	2:  (*Produktions Meldung*)
		Visu.MeldungProduktion.Color_R := 255;
		Visu.MeldungProduktion.Color_G := 255;
		Visu.MeldungProduktion.Color_B := 0;
		IF visu.s_akt_sprache = 'de' THEN
			Visu.MeldungProduktion.Name:='Y-Achse WT Übergabepos größer als Endlage';
		ELSIF visu.s_akt_sprache = 'en' THEN
			Visu.MeldungProduktion.Name:='Y-Achse WT Übergabepos größer als Endlage';
		ELSIF visu.s_akt_sprache = 'cz' THEN
			Visu.MeldungProduktion.Name:='Y-Achse WT Übergabepos größer als Endlage';
		END_IF
		Visu.MeldungProduktion.ShowMessage := TRUE;
		Visu.MeldungProduktion.Button1.sichtbar:= FALSE;	(*OK*)
		Visu.MeldungProduktion.Button1.Text:='Ok';
		i16_state_msg := 3;

	3:  (*Warte auf OK*)
		IF NOT b_EndlageErreicht THEN
			ST_Message_Produktion.b_PM_Quitt:=TRUE;
			i16_state_msg:=0;
		END_IF
END_CASE

(* =======================================Toplevel========================================== *)
(* Starte Inbetriebnahme-Sequenz *)
IF st_ctrl_in.b_gehe_step_ibn THEN
	fb_state_entry.i16_next_step := INBETRIEBNAHME;
END_IF

(* =====Achse wird disabled===== *)
IF (NOT e_steuerung_ein OR NOT e_ba_mit_bedingungen) AND y_achse.Status.Operational THEN
	st_drive_cmd.enu_cmd := POWER_DISABLE;
END_IF

IF fb_state_entry.i16_next_step > INIT AND fb_state_entry.i16_next_step < FEHLER THEN
	(* =====Fehler vom Achskontroller===== *)
	IF st_drive_cmd.b_job_fehler THEN
		fb_state_entry.i16_next_step := FEHLER;
	END_IF

	IF fb_state_entry.i16_next_step > 35 THEN
		(* Devicefehler *)
		IF y_achse.Status.Error THEN
			st_sm.b_achsfehler := TRUE;
			fb_state_entry.i16_next_step := FEHLER;
		ELSIF y_achse.Status.DriveDeviceError THEN
			st_sm.b_devicefehler := TRUE;
			fb_state_entry.i16_next_step := FEHLER;
		END_IF
	END_IF

	IF fb_state_entry.i16_next_step < STOP THEN
		(* =====Achse wird gestoppt===== *)
		IF st_ctrl_in.b_stop THEN
			fb_state_entry.i16_next_step := STOP;
		ELSIF fb_state_entry.i16_next_step < HALT THEN
			(* =====Achse wird angehalten===== *)
			IF st_ctrl_in.b_halt THEN
				fb_state_entry.i16_next_step := HALT;
			END_IF
		END_IF
	END_IF
END_IF

(* ======================================Schrittkette======================================== *)
fb_state_entry(
	i16_next_step:= ,
	i16_pos:= 1,
	E=> ,
	X=> , 
	i16_step=> ,
	i16_last_step=> );

CASE fb_state_entry.i16_step OF
(*=======================================================*)
	INIT_OBJ:
		IF st_config_achse.b_config_fertig THEN
			fb_state_entry.i16_next_step := 1;
		END_IF

(*=======================================================*)
	1:	(* Warte bis NetID´s der Slaves ausgelesen sind *)
		IF fb_state_entry.E THEN
			;
		END_IF

		(*-----------------------Weiterschaltbedingungen----------------------------*)
		IF ST_EthercatDiag.st_ctrl_out.b_fertig THEN
			fb_state_entry.i16_next_step := 2;
		END_IF

(*=======================================================*)
	2:	(* Spezifische NC-Achsparameter auslesen *)
		IF fb_state_entry.E THEN
			fb_axis.i16_nc_parameter_nummer := MaxVelocitySystem;
			st_drive_cmd.enu_cmd := READ_NC_PARAMETER;
		END_IF

		(*-----------------------Weiterschaltbedingungen----------------------------*)
		IF st_drive_cmd.enu_cmd = NO_COMMAND THEN
			lr_Velo_in:=st_geschwindigkeiten.lr_maximalgeschwindigkeit;
			st_geschwindigkeiten.lr_auto_max := st_geschwindigkeiten.lr_maximalgeschwindigkeit := fb_axis.r_wert_nc_read_parameter;
			st_geschwindigkeiten.lr_auto_min := 25.0;
			st_geschwindigkeiten.lr_jog := 50;
			fb_state_entry.i16_next_step := 3;
		END_IF

(*=======================================================*)
	3:	(* Spezifische NC-Achsparameter auslesen *)
		IF fb_state_entry.E THEN
			fb_axis.i16_nc_parameter_nummer := MaxAccelerationSystem;
			st_drive_cmd.enu_cmd := READ_NC_PARAMETER;
		END_IF

		(*-----------------------Weiterschaltbedingungen----------------------------*)
		IF st_drive_cmd.enu_cmd = NO_COMMAND THEN
			st_geschwindigkeiten.lr_beschleunigung := fb_axis.r_wert_nc_read_parameter;
			fb_state_entry.i16_next_step := 4;
		END_IF

(*=======================================================*)
	4:	(* Spezifische NC-Achsparameter auslesen *)
		IF fb_state_entry.E THEN
			fb_axis.i16_nc_parameter_nummer := MaxDecelerationSystem;
			st_drive_cmd.enu_cmd := READ_NC_PARAMETER;
		END_IF

		(*-----------------------Weiterschaltbedingungen----------------------------*)
		IF st_drive_cmd.enu_cmd = NO_COMMAND THEN
			st_geschwindigkeiten.lr_verzoegerung := fb_axis.r_wert_nc_read_parameter;
			lr_decceleration_normal := st_geschwindigkeiten.lr_verzoegerung;
			lr_decceleration_nothalt := 200000.0;
			fb_state_entry.i16_next_step := 5;
		END_IF

(*=======================================================*)
	5:	(* Spezifische NC-Achsparameter auslesen *)
		IF fb_state_entry.E THEN
			fb_axis.i16_nc_parameter_nummer := MaxJerk;
			st_drive_cmd.enu_cmd := READ_NC_PARAMETER;
		END_IF

		(*-----------------------Weiterschaltbedingungen----------------------------*)
		IF st_drive_cmd.enu_cmd = NO_COMMAND THEN
			st_geschwindigkeiten.lr_ruck := fb_axis.r_wert_nc_read_parameter;
			fb_state_entry.i16_next_step := 6;
		END_IF

(*=======================================================*)
	6:	(* Konfigurationen der Achse *)
		IF fb_state_entry.E THEN
			fb_axis.st_eccoe_sdo.s_ec_slave_net_id := ST_EthercatDiag.s_ec_slave_net_id[2];
			fb_axis.st_eccoe_sdo.ui16_slave_addr := st_config_achse.ui16_ethercat_adr;
		END_IF

		(*-----------------------Weiterschaltbedingungen----------------------------*)
		fb_state_entry.i16_next_step := 7;

(*=======================================================*)
	7:	(* Spezifische NC-Achsparameter auslesen *)
		IF fb_state_entry.E THEN
			fb_axis.i16_nc_parameter_nummer := AxisMinSoftPosLimit;
			st_drive_cmd.enu_cmd := READ_NC_PARAMETER;
		END_IF

		(*-----------------------Weiterschaltbedingungen----------------------------*)
		IF st_drive_cmd.enu_cmd = NO_COMMAND THEN
			lr_MinSoftPosLimit := fb_axis.r_wert_nc_read_parameter;
			fb_state_entry.i16_next_step := 8;
		END_IF


(*=======================================================*)
	8:	(* Spezifische NC-Achsparameter auslesen *)
		IF fb_state_entry.E THEN
			fb_axis.i16_nc_parameter_nummer := AxisMaxSoftPosLimit;
			st_drive_cmd.enu_cmd := READ_NC_PARAMETER;
		END_IF

		(*-----------------------Weiterschaltbedingungen----------------------------*)
		IF st_drive_cmd.enu_cmd = NO_COMMAND THEN
			lr_MaxSoftPosLimit := fb_axis.r_wert_nc_read_parameter;
			fb_state_entry.i16_next_step := FEHLER; (*in Fehler gehen damit die Achsen resetet werden. Sonst steigen die Achsen bei einem TC Restart aus*)
		END_IF

(*=======================================================*)
	INIT:
		IF fb_state_entry.E THEN
			fb_ton_wz.IN := FALSE;
			fb_ton_uez.IN	:= FALSE;
			fb_ton_quitt.IN := FALSE;
			(* Reset Stoermeldungen *)
			st_sm.b_achse_nicht_auf_startpos := FALSE;
			st_sm.b_achsfehler := FALSE;
			st_sm.b_devicefehler := FALSE;
			st_sm.b_keine_verfahrfreigabe := FALSE;
			st_sm.b_ende_skalierungs_nocke := FALSE;
			st_sm.b_ende_camming_nocke := FALSE;
			st_sm.b_skalierung_noch_aktiv := FALSE;
			b_start_in:=FALSE;
			st_ctrl_out.b_busy:=FALSE;
			st_ctrl_out.b_fehler := FALSE;
			st_ctrl_out.b_fertig := FALSE;

			st_ctrl_out.b_bereit := FALSE;
			st_ctrl_out.b_prebereit := FALSE;
			sm_kein_nocken_definiert := FALSE;

			fb_axis.lr_soll_geschwindigkeit := gst_datensatz.st_wkz.r_auto_y;

			st_geschwindigkeiten.lr_verzoegerung := lr_decceleration_normal;
		END_IF

		(*-----------------------Weiterschaltbedingungen----------------------------*)
		IF st_ctrl_in.b_preinit THEN
			fb_state_entry.i16_next_step := 15;
		END_IF

(*=======================================================*)
	15:	(* Reglerfreigabe wegnehmen *)
		IF fb_state_entry.E THEN
			st_drive_cmd.enu_cmd := POWER_DISABLE;
		END_IF

		(*-----------------------Weiterschaltbedingungen----------------------------*)
		IF st_drive_cmd.enu_cmd = NO_COMMAND THEN
			fb_state_entry.i16_next_step := 20;
		END_IF

(*=======================================================*)
	20:	(* Überprüfe Nullpunktverschiebung des Absolutwertgebers auf Korrektheit *)
		IF fb_state_entry.E THEN
			fb_axis.i16_nc_parameter_nummer := AxisEncoderOffset;	(* vom Datentyp MC_AxisParameter *)
			st_drive_cmd.enu_cmd := READ_NC_PARAMETER;
		END_IF

		(*-----------------------Weiterschaltbedingungen----------------------------*)
		IF st_drive_cmd.enu_cmd = NO_COMMAND THEN
			IF fb_axis.r_wert_nc_read_parameter = gst_datensatz.st_md.st_md_y_achse.lr_nullpunktverschiebung THEN
				fb_state_entry.i16_next_step := 35;	(* Reglerfreigabe setzen *)
			ELSE
				fb_state_entry.i16_next_step := 25;	(* Nullpunktverschiebung schreiben *)
			END_IF
		END_IF

(*=======================================================*)
	25:	(* Nullpunktverschiebung hat sich geändert, deshalb erst Null reinschreiben, um keinen Additionsfehler zu machen, *)
		(* weil der Wert der Verschiebung beim Neustart komplett auf die Achse geschrieben wird *)
		IF fb_state_entry.E THEN
			fb_axis.i16_nc_parameter_nummer := AxisEncoderOffset;
			fb_axis.r_wert_nc_write_parameter := 0.0;
			st_drive_cmd.enu_cmd := WRITE_NC_PARAMETER;
		END_IF

		(*-----------------------Weiterschaltbedingungen----------------------------*)
		IF st_drive_cmd.enu_cmd = NO_COMMAND THEN
			fb_state_entry.i16_next_step := 30;
		END_IF

(*=======================================================*)
	30:	(* Aktuelle Nullpunktverschiebung des Absolutwertgebers an die Achse senden *)
		IF fb_state_entry.E THEN
			fb_axis.i16_nc_parameter_nummer := AxisEncoderOffset;
			fb_axis.r_wert_nc_write_parameter := gst_datensatz.st_md.st_md_y_achse.lr_nullpunktverschiebung;
			st_drive_cmd.enu_cmd := WRITE_NC_PARAMETER;
		END_IF

		(*-----------------------Weiterschaltbedingungen----------------------------*)
		IF st_drive_cmd.enu_cmd = NO_COMMAND THEN
			fb_state_entry.i16_next_step := 35;
		END_IF

(*=======================================================*)
	35:	(* Reglerfreigabe setzen , Reset wird bei Bedarf automatisch ausgeführt*)
		IF fb_state_entry.E THEN
			st_drive_cmd.enu_cmd := POWER_ENABLE;
		END_IF

		(*-----------------------Weiterschaltbedingungen----------------------------*)
		IF st_drive_cmd.enu_cmd = NO_COMMAND THEN
			fb_state_entry.i16_next_step := 40;
		END_IF

(*=======================================================*)
	40:	(* Nullpunktverschiebung ist geschrieben *)
		IF fb_state_entry.E THEN
			st_ctrl_out.b_prebereit := TRUE;
		END_IF

		(*-----------------------Weiterschaltbedingungen----------------------------*)
		IF st_ctrl_in.b_init THEN
			fb_state_entry.i16_next_step := 45;
		END_IF

(*=======================================================*)
	45: (* Warte auf Startsignal zum Positionieren *)

		(*-----------------------Weiterschaltbedingungen----------------------------*)
		IF st_ctrl_in.b_start THEN
			fb_state_entry.i16_next_step := 50;
		END_IF

(*=======================================================*)
	50: (* Positioniere Achse auf ausgelesene Slaveposition *)
		IF fb_state_entry.E THEN
			fb_axis.st_position.r_soll := ST_Z_Achse.lr_slave_position;
			st_drive_cmd.enu_cmd := MOVE_ABSOLUTE;
		END_IF

		(*-----------------------Weiterschaltbedingungen----------------------------*)
		IF st_drive_cmd.enu_cmd = NO_COMMAND THEN
			fb_state_entry.i16_next_step := 60;
		END_IF

(*=======================================================*)
	60: (* Warte bis Y-Achse gekoppelt wurde *)
		IF fb_state_entry.E THEN
			st_ctrl_out.b_fertig := TRUE;
		END_IF

		(*-----------------------Weiterschaltbedingungen----------------------------*)
		IF y_achse.NcToPlc.CoupleState = 3 THEN
			st_ctrl_out.b_fertig := FALSE;
			fb_state_entry.i16_next_step := BEREIT;
		END_IF

(*=======================================================*)
	BEREIT:
		IF fb_state_entry.E THEN
			st_ctrl_out.b_bereit := TRUE;
			enu_cmd_in:=NO_COMMAND;
		END_IF

		(*-----------------------Weiterschaltbedingungen----------------------------*)
		IF fb_r_trig_start.Q THEN
			st_ctrl_out.b_fertig_2 := FALSE;
			fb_state_entry.i16_next_step := 110;
		END_IF

		IF 	fb_r_trig_start_in.Q THEN		(*neu! zum Starten einer Positionierung von einem externen Prg.*)
			st_ctrl_out.b_fertig := FALSE;
			fb_state_entry.i16_next_step := 102;
		END_IF

		IF fb_state_entry.X THEN
			st_ctrl_out.b_fertig := FALSE;
			st_ctrl_out.b_busy:=TRUE;
		END_IF

(*=======================================================*)
	102:
		IF 	fb_state_entry.E THEN
			b_start_in:=FALSE;
		END_IF

		(*-----------------------Weiterschaltbedingungen----------------------------*)
		IF 	st_drive_cmd.enu_cmd = NO_COMMAND THEN
			fb_state_entry.i16_next_step := 104;
		END_IF

(*=======================================================*)
	104: (* Positioniere Achse  *)
		IF 	fb_state_entry.E THEN
			fb_axis.st_position.r_soll := lr_Achspos_in ;
			fb_axis.lr_soll_geschwindigkeit:=lr_Velo_in;
			st_drive_cmd.enu_cmd := enu_cmd_in;
		END_IF

		(*-----------------------Weiterschaltbedingungen----------------------------*)
		IF 	st_drive_cmd.enu_cmd = NO_COMMAND THEN
			st_ctrl_out.b_fertig := TRUE;
			fb_state_entry.i16_next_step := BEREIT;
		END_IF

		IF 	fb_state_entry.X THEN
			st_ctrl_out.b_busy:=FALSE;
		END_IF

(*=======================================================*)
	110: (* Fallunterscheidung *)
		CASE gst_datensatz.st_md.i16_typ_zelle OF
			KEINE_ZELLE:
				;

			BESTUECKZELLE_1700:
				(*-----------------------Weiterschaltbedingungen----------------------------*)
				fb_state_entry.i16_next_step := 200;

			RASTERFOLIE:
				(*-----------------------Weiterschaltbedingungen----------------------------*)
				fb_state_entry.i16_next_step := 120;

		END_CASE

(*=======================================================*)
	120: (* Positioniere Achse auf  0-Koordinate  des ISK *)
		IF fb_state_entry.E THEN
			fb_axis.st_position.r_soll := 	gst_datensatz.st_isk.lr_pos_y_0 +
										gst_datensatz.st_wkz.lr_offset_y_pos_0 +
										gst_datensatz.st_wt.lr_offset_y_pos_0 +
										gst_datensatz.st_md.lr_offset_y_pos_0 +
										gst_datensatz.st_bestueckprogramm.lr_y[0];
			st_drive_cmd.enu_cmd := MOVE_ABSOLUTE;
		END_IF

		(*-----------------------Weiterschaltbedingungen----------------------------*)
		IF st_drive_cmd.enu_cmd = NO_COMMAND THEN
			st_ctrl_out.b_fertig := TRUE;
			st_ctrl_out.b_busy:=FALSE;
			fb_state_entry.i16_next_step := 300;
		END_IF

(*=======================================================*)
	200:
		IF fb_state_entry.E THEN
			st_ctrl_out.b_fertig := TRUE;
			st_ctrl_out.b_busy:=FALSE;
		END_IF

		(*-----------------------Weiterschaltbedingungen----------------------------*)
		IF st_ctrl_in.b_start_2 THEN
			st_ctrl_out.b_fertig := FALSE;
			fb_state_entry.i16_next_step := 210;
		END_IF

(*=======================================================*)
	210: (* Positioniere Achse auf gewünschte Position *)
		IF fb_state_entry.E THEN
			fb_axis.st_position.r_soll :=  ST_Z_Achse.lr_slave_position;
			st_drive_cmd.enu_cmd := MOVE_ABSOLUTE;
		END_IF

		(*-----------------------Weiterschaltbedingungen----------------------------*)
		IF st_drive_cmd.enu_cmd = NO_COMMAND THEN
			fb_state_entry.i16_next_step := 220;
		END_IF

(*=======================================================*)
	220: (* Warte bis Y-Achse gekoppelt wurde *)
		IF fb_state_entry.E THEN
			st_ctrl_out.b_fertig_2 := TRUE;
		END_IF

		(*-----------------------Weiterschaltbedingungen----------------------------*)
		IF y_achse.NcToPlc.CoupleState = 3 THEN
			st_ctrl_out.b_fertig_2 := FALSE;
			fb_state_entry.i16_next_step := BEREIT;
		END_IF

(*=======================================================*)
	300:(* Verfahre Y-Achse undwarte auf Start von Z-Achse *)

		(*-----------------------Weiterschaltbedingungen----------------------------*)
		(* Verfahre Y-Achse *)
		IF	gst_datensatz.st_md.i16_typ_zelle = RASTERFOLIE AND
			ST_Rasterfolienmontage.b_start_y_Achse THEN
			fb_state_entry.i16_next_step := 310;
		END_IF

		(* Warte auf Start von Z-Achse *)
		IF st_ctrl_in.b_start_2 THEN
			st_ctrl_out.b_fertig := FALSE;
			fb_state_entry.i16_next_step := 350;
		END_IF

(*=======================================================*)
	310: (* Positioniere Achse  *)
		IF fb_state_entry.E THEN
			fb_axis.st_position.r_soll := 	lr_tmp_Achspos;
			st_drive_cmd.enu_cmd := MOVE_ABSOLUTE;
		END_IF

		(*-----------------------Weiterschaltbedingungen----------------------------*)
		IF st_drive_cmd.enu_cmd = NO_COMMAND THEN
			fb_state_entry.i16_next_step := 300;
			ST_Rasterfolienmontage.b_start_y_Achse:=FALSE;
		END_IF


(*=======================================================*)
	350: (* Positioniere Achse auf gewünschte Position am Ende der Kurvenscheibe *)
		IF fb_state_entry.E THEN
			fb_axis.st_position.r_soll :=  ST_Z_Achse.lr_slave_position;
			st_drive_cmd.enu_cmd := MOVE_ABSOLUTE;
		END_IF

		(*-----------------------Weiterschaltbedingungen----------------------------*)
		IF st_drive_cmd.enu_cmd = NO_COMMAND THEN
			fb_state_entry.i16_next_step := 360;
		END_IF

(*=======================================================*)
	360: (* Warte bis Y-Achse gekoppelt wurde *)
		IF fb_state_entry.E THEN
			st_ctrl_out.b_fertig_2 := TRUE;
		END_IF

		(*-----------------------Weiterschaltbedingungen----------------------------*)
		IF y_achse.NcToPlc.CoupleState = 3 THEN
			st_ctrl_out.b_fertig_2 := FALSE;
			fb_state_entry.i16_next_step := BEREIT;
		END_IF

(*=======================================================*)
	FEHLER:
		IF fb_state_entry.E THEN
			st_ctrl_out.b_fehler := TRUE;
			fb_ton_quitt.IN := FALSE;
			st_ctrl_out.b_busy:=FALSE;
		END_IF

		IF st_ctrl_in.b_stop AND NOT y_achse.Status.HasBeenStopped THEN
			st_drive_cmd.enu_cmd := STOP_AXIS;
		END_IF

		IF st_ctrl_in.b_halt AND y_achse.Status.Moving THEN
			st_drive_cmd.enu_cmd := HALT_AXIS;
			st_geschwindigkeiten.lr_verzoegerung := lr_decceleration_nothalt;
		END_IF

		(*-----------------------Weiterschaltbedingungen----------------------------*)
		IF st_ctrl_in.b_quitt AND NOT fb_state_entry.E THEN
			st_ctrl_out.b_fehler := FALSE;
			st_drive_cmd.enu_cmd := RESET;
			fb_ton_quitt.IN := TRUE;
		END_IF

		IF fb_ton_quitt.Q THEN
			fb_ton_quitt.IN := FALSE;
			fb_state_entry.i16_next_step := INIT;
		END_IF

(*=======================================================*)
	STOP:
		IF fb_state_entry.E THEN
			st_ctrl_out.b_busy:=FALSE;
			IF y_achse.NcToPlc.CoupleState = 0 THEN
				st_drive_cmd.enu_cmd := STOP_AXIS;
			END_IF
		END_IF

		(*-----------------------Weiterschaltbedingungen----------------------------*)
		IF st_drive_cmd.enu_cmd = NO_COMMAND AND y_achse.Status.NotMoving THEN
			fb_state_entry.i16_next_step := STILLSTAND;
		END_IF

(*=======================================================*)
	STILLSTAND:
		IF fb_state_entry.E THEN
			st_drive_cmd.enu_cmd := POWER_DISABLE;
			fb_ton_quitt.IN := FALSE;
		END_IF

		(*-----------------------Weiterschaltbedingungen----------------------------*)
		IF st_ctrl_in.b_quitt AND NOT fb_state_entry.E THEN
			fb_ton_quitt.IN := TRUE;
		END_IF

		IF fb_ton_quitt.Q THEN
			fb_ton_quitt.IN := FALSE;
			fb_state_entry.i16_next_step := INIT;
		END_IF

(*=======================================================*)
	HALT:
		IF fb_state_entry.E THEN
			IF y_achse.NcToPlc.CoupleState = 0 THEN
				st_drive_cmd.enu_cmd := HALT_AXIS;
				st_geschwindigkeiten.lr_verzoegerung := lr_decceleration_nothalt;
			END_IF
			fb_ton_quitt.IN := FALSE;
		END_IF

		(*-----------------------Weiterschaltbedingungen----------------------------*)
		IF st_ctrl_in.b_quitt AND NOT fb_state_entry.E THEN
			fb_ton_quitt.IN := TRUE;
		END_IF

		IF fb_ton_quitt.Q THEN
			fb_ton_quitt.IN := FALSE;
			fb_state_entry.i16_next_step := INIT;
		END_IF

(*=======================================================*)
	HANDRAD:	(* Überprüfe Nullpunktverschiebung des Absolutwertgebers auf Korrektheit *)
		IF fb_state_entry.E THEN
			st_ctrl_out.b_fehler := TRUE;
			fb_axis.i16_nc_parameter_nummer := AxisEncoderOffset;
			st_drive_cmd.enu_cmd := READ_NC_PARAMETER;
		END_IF

		(*-----------------------Weiterschaltbedingungen----------------------------*)
		IF st_drive_cmd.enu_cmd = NO_COMMAND THEN
			IF fb_axis.r_wert_nc_read_parameter = gst_datensatz.st_md.st_md_y_achse.lr_nullpunktverschiebung THEN
				fb_state_entry.i16_next_step := 2040;	(* Jogbetrieb *)
			ELSE
				fb_state_entry.i16_next_step := 2010;	(* Reglerfreigabe nehmen und Nullpunktverschiebung schreiben *)
			END_IF
		END_IF

(*=======================================================*)
	2010:	(* Reglerfreigabe wegnehmen , damit Nullpunktverschiebung geschrieben werden kannt*)
		IF fb_state_entry.E THEN
			st_drive_cmd.enu_cmd := POWER_DISABLE;
		END_IF

		(*-----------------------Weiterschaltbedingungen----------------------------*)
		IF st_drive_cmd.enu_cmd = NO_COMMAND THEN
			fb_state_entry.i16_next_step := 2020;
		END_IF

(*=======================================================*)
	2020:	(* Nullpunktverschiebung hat sich geändert, deshalb erst Null reinschreiben, um keinen Additionsfehler zu machen, *)
			(* weil der Wert der Verschiebung beim Neustart komplett auf die Achse geschrieben wird *)
		IF fb_state_entry.E THEN
			fb_axis.i16_nc_parameter_nummer := AxisEncoderOffset;
			fb_axis.r_wert_nc_write_parameter := 0.0;
			st_drive_cmd.enu_cmd := WRITE_NC_PARAMETER;
		END_IF

		(*-----------------------Weiterschaltbedingungen----------------------------*)
		IF st_drive_cmd.enu_cmd = NO_COMMAND THEN
			fb_state_entry.i16_next_step := 2030;
		END_IF

(*=======================================================*)
	2030:	(* Aktuelle Nullpunktverschiebung des Absolutwertgebers an die Achse senden *)
		IF fb_state_entry.E THEN
			fb_axis.i16_nc_parameter_nummer := AxisEncoderOffset;
			fb_axis.r_wert_nc_write_parameter := gst_datensatz.st_md.st_md_y_achse.lr_nullpunktverschiebung;
			st_drive_cmd.enu_cmd := WRITE_NC_PARAMETER;
		END_IF

		(*-----------------------Weiterschaltbedingungen----------------------------*)
		IF st_drive_cmd.enu_cmd = NO_COMMAND THEN
			fb_state_entry.i16_next_step := 2040;
		END_IF

(*=======================================================*)
	2040:	(* Jogbetrieb *)
		IF fb_state_entry.E THEN
			fb_axis.lr_soll_geschwindigkeit := st_geschwindigkeiten.lr_jog;
		END_IF

		IF ST_Euchner_Handbedienpult.i16_Handrad_delta > 0 THEN
			st_drive_cmd.enu_cmd := JOG_VORWAERTS;
		ELSIF ST_Euchner_Handbedienpult.i16_Handrad_delta < 0 THEN
			st_drive_cmd.enu_cmd := JOG_RUECKWAERTS;
		ELSIF  y_achse.Status.Moving THEN
			st_drive_cmd.enu_cmd := JOG_STOP;
		END_IF

		IF fb_r_trig_taste_plus.Q THEN
			fb_state_entry.i16_next_step := MOTORBREMSE_AUF;
		END_IF
		IF fb_r_trig_taste_minus.Q THEN
			fb_state_entry.i16_next_step := MOTORBREMSE_ZU;
		END_IF

		(*-----------------------Weiterschaltbedingungen----------------------------*)
		IF gi16_betriebsart <> HAND OR NOT b_hand_dialog_aktiv THEN
			fb_state_entry.i16_next_step := 2050;
		END_IF

(*=======================================================*)
	2050:
		IF fb_state_entry.E THEN
			st_drive_cmd.enu_cmd := ABORT;
		END_IF

		(*-----------------------Weiterschaltbedingungen----------------------------*)
		IF st_drive_cmd.enu_cmd = NO_COMMAND THEN
			fb_state_entry.i16_next_step := 2060;
		END_IF

(*=======================================================*)
	2060:
		IF fb_state_entry.E THEN
			fb_axis.w_idn := P_0_IDN + 96;
			fb_axis.ui16_soeparam_write_value := 0;	(* Motorbremse im Automatikbetrieb für reguläres Fahren *)
			st_drive_cmd.enu_cmd := SOE_WRITE_PARAM;
		END_IF

		(*-----------------------Weiterschaltbedingungen----------------------------*)
		IF st_drive_cmd.enu_cmd = NO_COMMAND THEN
			fb_state_entry.i16_next_step := 2070;
		END_IF

(*=======================================================*)
	2070:	(* Reglerfreigabe wegnehmen *)
		IF fb_state_entry.E THEN
			st_drive_cmd.enu_cmd := POWER_DISABLE;
		END_IF

		(*-----------------------Weiterschaltbedingungen----------------------------*)
		IF st_drive_cmd.enu_cmd = NO_COMMAND THEN
			st_ctrl_out.b_fehler := FALSE;
			fb_state_entry.i16_next_step := INIT;
		END_IF

(*=======================================================*)
	MOTORBREMSE_AUF:
		IF fb_state_entry.E THEN
			st_drive_cmd.enu_cmd := ABORT;
		END_IF

		(*-----------------------Weiterschaltbedingungen----------------------------*)
		IF st_drive_cmd.enu_cmd = NO_COMMAND THEN
			fb_state_entry.i16_next_step := 2110;
		END_IF

(*=======================================================*)
	2110:	(* Reglerfreigabe wegnehmen *)
		IF fb_state_entry.E THEN
			st_drive_cmd.enu_cmd := POWER_DISABLE;
		END_IF

		(*-----------------------Weiterschaltbedingungen----------------------------*)
		IF st_drive_cmd.enu_cmd = NO_COMMAND THEN
			fb_state_entry.i16_next_step := 2120;
		END_IF

(*=======================================================*)
	2120:	(* Bremse auf machen *)
		IF fb_state_entry.E THEN
			fb_axis.w_idn := P_0_IDN + 96;
			fb_axis.ui16_soeparam_write_value := 2;
			st_drive_cmd.enu_cmd := SOE_WRITE_PARAM;
		END_IF

		(*-----------------------Weiterschaltbedingungen----------------------------*)
		IF 	st_drive_cmd.enu_cmd = NO_COMMAND AND
			(gi16_betriebsart <> HAND OR
			NOT b_hand_dialog_aktiv OR
			ST_Euchner_Handbedienpult.i16_Handrad_delta > 0)
			THEN
				fb_state_entry.i16_next_step := HANDRAD;
		ELSIF fb_r_trig_taste_minus.Q THEN
			fb_state_entry.i16_next_step := MOTORBREMSE_ZU;
		END_IF

(*=======================================================*)
	MOTORBREMSE_ZU:
		IF fb_state_entry.E THEN
			st_drive_cmd.enu_cmd := ABORT;
		END_IF

		(*-----------------------Weiterschaltbedingungen----------------------------*)
		IF st_drive_cmd.enu_cmd = NO_COMMAND THEN
			fb_state_entry.i16_next_step := 2210;
		END_IF

(*=======================================================*)
	2210:	(* Reglerfreigabe setzen *)
		IF fb_state_entry.E THEN
			st_drive_cmd.enu_cmd := POWER_ENABLE;
		END_IF

		(*-----------------------Weiterschaltbedingungen----------------------------*)
		IF st_drive_cmd.enu_cmd = NO_COMMAND THEN
			fb_state_entry.i16_next_step := 2220;
		END_IF

(*=======================================================*)
	2220:	(* Bremse zu machen *)
		IF fb_state_entry.E THEN
			fb_axis.w_idn := P_0_IDN + 96;
			fb_axis.ui16_soeparam_write_value := 0;
			st_drive_cmd.enu_cmd := SOE_WRITE_PARAM;
		END_IF

		(*-----------------------Weiterschaltbedingungen----------------------------*)
		IF 	st_drive_cmd.enu_cmd = NO_COMMAND AND
			(gi16_betriebsart <> HAND OR
			NOT b_hand_dialog_aktiv OR
			ST_Euchner_Handbedienpult.i16_Handrad_delta > 0)
			THEN
				fb_state_entry.i16_next_step := HANDRAD;
		ELSIF fb_r_trig_taste_plus.Q THEN
			fb_state_entry.i16_next_step := MOTORBREMSE_AUF;
		END_IF

(*=======================================================*)
	NULLPUNKT_SETZEN:
		(* Aktuellen Jog beenden, sonst Probleme beim Softwareendschalter*)
		IF fb_state_entry.E THEN
			st_drive_cmd.enu_cmd := JOG_STOP;
		END_IF

		(*-----------------------Weiterschaltbedingungen----------------------------*)
		IF st_drive_cmd.enu_cmd = NO_COMMAND THEN
			fb_state_entry.i16_next_step := 2505;
		END_IF

(*=======================================================*)
	2505:
		(* 	Lese aktuelle Nullpunkt verschiebung von der Hardware. Der Benutze könnte einen falschen
			Wert eingetragen haben *)
		IF fb_state_entry.E THEN
			fb_axis.i16_nc_parameter_nummer := AxisEncoderOffset;
			st_drive_cmd.enu_cmd := READ_NC_PARAMETER;
		END_IF

		(*-----------------------Weiterschaltbedingungen----------------------------*)
		IF st_drive_cmd.enu_cmd = NO_COMMAND THEN
			gst_datensatz.st_md.st_md_y_achse.lr_nullpunktverschiebung := fb_axis.r_wert_nc_read_parameter;
			fb_state_entry.i16_next_step := 2510;
		END_IF

(*=======================================================*)
	2510:	(* Nullpunktverschiebung berechnen *)
		IF fb_state_entry.E THEN
			lr_pos_ohneverschiebung := axis_y_achse.st_visu.lr_position_ist - gst_datensatz.st_md.st_md_y_achse.lr_nullpunktverschiebung;

			gst_datensatz.st_md.st_md_y_achse.lr_nullpunktverschiebung := - lr_pos_ohneverschiebung;
		END_IF

		(*-----------------------Weiterschaltbedingungen----------------------------*)
		(* Aktiviere den wert in die Hardware *)
		fb_state_entry.i16_next_step := HANDRAD;

(*=======================================================*)
	INBETRIEBNAHME:	(* Überprüfe Nullpunktverschiebung des Absolutwertgebers auf Korrektheit *)
		IF fb_state_entry.E THEN
			fb_axis.i16_nc_parameter_nummer := AxisEncoderOffset;
			st_drive_cmd.enu_cmd := READ_NC_PARAMETER;
		END_IF

		(*-----------------------Weiterschaltbedingungen----------------------------*)
		IF st_drive_cmd.enu_cmd = NO_COMMAND THEN
			IF fb_axis.r_wert_nc_read_parameter = gst_datensatz.st_md.st_md_y_achse.lr_nullpunktverschiebung THEN
				fb_state_entry.i16_next_step := 5100;	(* Reversiersequenz*)
			ELSE
				fb_state_entry.i16_next_step := 5010;	(* Reglerfreigabe nehmen und Nullpunktverschiebung schreiben *)
			END_IF
		END_IF

(*=======================================================*)
	5010:	(* Reglerfreigabe wegnehmen, damit Nullpunktverschiebung geschrieben werden kannt*)
		IF fb_state_entry.E THEN
			st_drive_cmd.enu_cmd := POWER_DISABLE;
		END_IF

		(*-----------------------Weiterschaltbedingungen----------------------------*)
		IF st_drive_cmd.enu_cmd = NO_COMMAND THEN
			fb_state_entry.i16_next_step := 5020;
		END_IF

(*=======================================================*)
	5020:	(* Nullpunktverschiebung hat sich geändert, deshalb erst Null reinschreiben, um keinen Additionsfehler zu machen, *)
			(* weil der Wert der Verschiebung beim Neustart komplett auf die Achse geschrieben wird *)
		IF fb_state_entry.E THEN
			fb_axis.i16_nc_parameter_nummer := AxisEncoderOffset;
			fb_axis.r_wert_nc_write_parameter := 0.0;
			st_drive_cmd.enu_cmd := WRITE_NC_PARAMETER;
		END_IF

		(*-----------------------Weiterschaltbedingungen----------------------------*)
		IF st_drive_cmd.enu_cmd = NO_COMMAND THEN
			fb_state_entry.i16_next_step := 5030;
		END_IF

(*=======================================================*)
	5030:	(* Aktuelle Nullpunktverschiebung des Absolutwertgebers an die Achse senden *)
		IF fb_state_entry.E THEN
			fb_axis.i16_nc_parameter_nummer := AxisEncoderOffset;
			fb_axis.r_wert_nc_write_parameter := gst_datensatz.st_md.st_md_y_achse.lr_nullpunktverschiebung;
			st_drive_cmd.enu_cmd := WRITE_NC_PARAMETER;
		END_IF

		(*-----------------------Weiterschaltbedingungen----------------------------*)
		IF st_drive_cmd.enu_cmd = NO_COMMAND THEN
			fb_state_entry.i16_next_step := 5100;
		END_IF

(*=======================================================*)
	5100:	(* Verfahren der Achse zwischen zwei Punkten zum Testen verschiedener Achsparameter *)
		IF fb_state_entry.E THEN
			fb_axis.lr_soll_geschwindigkeit := st_geschwindigkeiten.lr_jog;
			fb_axis.st_position.lr_ibn_pos_start := 0.0;
			fb_axis.st_position.lr_ibn_pos_ziel := 25.0;
		END_IF

		(*-----------------------Weiterschaltbedingungen----------------------------*)
		IF st_ctrl_in.b_ibn_start THEN
			fb_state_entry.i16_next_step := 5110;
		END_IF

(*=======================================================*)
	5110: (* Fahre Y-Achse auf Startposition *)
(*
		IF fb_state_entry.E THEN
			 fb_axis.st_position.r_soll := fb_axis.st_position.lr_ibn_pos_start;
			st_drive_cmd.enu_cmd := MOVE_ABSOLUTE;
		END_IF

		(*-----------------------Weiterschaltbedingungen----------------------------*)
		IF st_drive_cmd.enu_cmd = NO_COMMAND THEN
			fb_state_entry.i16_next_step := 5120;
		END_IF
*)
		IF fb_state_entry.E THEN
			st_drive_cmd.enu_cmd := POWER_ENABLE;
		END_IF

		(*-----------------------Weiterschaltbedingungen----------------------------*)
		IF st_drive_cmd.enu_cmd = NO_COMMAND THEN
			;
		END_IF

(*=======================================================*)
	5120: (* Pause *)
		IF fb_state_entry.E THEN
			fb_ton_wz.PT := t#1s;
			fb_ton_wz.IN := TRUE;
		END_IF

		(*-----------------------Weiterschaltbedingungen----------------------------*)
		IF fb_ton_wz.Q THEN
			fb_ton_wz.IN := FALSE;
			fb_state_entry.i16_next_step := 5130;
		END_IF

(*=======================================================*)
	5130: (* Fahre Z-Achse auf Zielposition *)
		IF fb_state_entry.E THEN
			 fb_axis.st_position.r_soll := fb_axis.st_position.lr_ibn_pos_ziel;
			st_drive_cmd.enu_cmd := MOVE_ABSOLUTE;
		END_IF

		(*-----------------------Weiterschaltbedingungen----------------------------*)
		IF st_drive_cmd.enu_cmd = NO_COMMAND THEN
			fb_state_entry.i16_next_step := 5140;
		END_IF

(*=======================================================*)
	5140: (* Pause *)
		IF fb_state_entry.E THEN
			fb_ton_wz.PT := t#1s;
			fb_ton_wz.IN := TRUE;
		END_IF

		(*-----------------------Weiterschaltbedingungen----------------------------*)
		IF fb_ton_wz.Q THEN
			fb_ton_wz.IN := FALSE;
			fb_state_entry.i16_next_step := 5100;
		END_IF
END_CASE

fb_state_entry(
	i16_next_step:= , 
	i16_pos:= 2,
	s_debugtext:= ,
	E=> ,
	X=> ,
	i16_step=> ,
	i16_last_step=> );

IF st_config_achse.b_config_fertig THEN
	(* Fehlermeldungen und Betriebsmeldungen ab dem Startindex in die globalen Meldungsarrays schreiben *)
	garr_stoermeldungen[st_config_achse.i16_meld_startindex + 0] := st_sm.b_achse_nicht_bb;
	garr_stoermeldungen[st_config_achse.i16_meld_startindex + 1] := st_sm.b_achse_nicht_referenziert;
	garr_stoermeldungen[st_config_achse.i16_meld_startindex + 2] := st_sm.b_keine_verfahrfreigabe;
	garr_stoermeldungen[st_config_achse.i16_meld_startindex + 3] := st_sm.b_achse_nicht_auf_startpos;
	garr_stoermeldungen[st_config_achse.i16_meld_startindex + 4] := st_sm.b_ende_skalierungs_nocke;
	garr_stoermeldungen[st_config_achse.i16_meld_startindex + 5] := st_sm.b_ende_camming_nocke;
	garr_stoermeldungen[st_config_achse.i16_meld_startindex + 6] := st_sm.b_skalierung_noch_aktiv;
	garr_stoermeldungen[st_config_achse.i16_meld_startindex + 7] := FALSE;
	garr_stoermeldungen[st_config_achse.i16_meld_startindex + 8] := FALSE;
	garr_stoermeldungen[st_config_achse.i16_meld_startindex + 9] := FALSE;
	garr_stoermeldungen[st_config_achse.i16_meld_startindex + 10] := sm_kein_nocken_definiert;
	garr_stoermeldungen[st_config_achse.i16_meld_startindex + 11] := FALSE;
	garr_stoermeldungen[st_config_achse.i16_meld_startindex + 12] := FALSE;
	garr_stoermeldungen[st_config_achse.i16_meld_startindex + 13] := FALSE;
	garr_stoermeldungen[st_config_achse.i16_meld_startindex + 14] := FALSE;
	garr_stoermeldungen[st_config_achse.i16_meld_startindex + 15] := FALSE;
	garr_stoermeldungen[st_config_achse.i16_meld_startindex + 16] := st_drive_cmd.meldungen.sm_write_soe_parameter;
	garr_stoermeldungen[st_config_achse.i16_meld_startindex + 17] := st_drive_cmd.meldungen.sm_read_soe_parameter;
	garr_stoermeldungen[st_config_achse.i16_meld_startindex + 18] := st_drive_cmd.meldungen.sm_write_nc_parameter;
	garr_stoermeldungen[st_config_achse.i16_meld_startindex + 19] := st_drive_cmd.meldungen.sm_read_nc_parameter;
	garr_stoermeldungen[st_config_achse.i16_meld_startindex + 20] := st_drive_cmd.meldungen.sm_power_enable;
	garr_stoermeldungen[st_config_achse.i16_meld_startindex + 21] := st_drive_cmd.meldungen.sm_power_disable;
	garr_stoermeldungen[st_config_achse.i16_meld_startindex + 22] := st_drive_cmd.meldungen.sm_reset;
	garr_stoermeldungen[st_config_achse.i16_meld_startindex + 23] := st_drive_cmd.meldungen.sm_home;
	garr_stoermeldungen[st_config_achse.i16_meld_startindex + 24] := st_drive_cmd.meldungen.sm_setposition;
	garr_stoermeldungen[st_config_achse.i16_meld_startindex + 25] := st_drive_cmd.meldungen.sm_jog_vorwaerts;
	garr_stoermeldungen[st_config_achse.i16_meld_startindex + 26] := st_drive_cmd.meldungen.sm_jog_rueckwaerts;
	garr_stoermeldungen[st_config_achse.i16_meld_startindex + 27] := st_drive_cmd.meldungen.sm_move_absolute;
	garr_stoermeldungen[st_config_achse.i16_meld_startindex + 28] := st_drive_cmd.meldungen.sm_move_relative;
	garr_stoermeldungen[st_config_achse.i16_meld_startindex + 29] := st_drive_cmd.meldungen.sm_move_velocity;
	garr_stoermeldungen[st_config_achse.i16_meld_startindex + 30] := st_drive_cmd.meldungen.sm_move_modulo;
	garr_stoermeldungen[st_config_achse.i16_meld_startindex + 31] := st_drive_cmd.meldungen.sm_stop_axis;
	garr_stoermeldungen[st_config_achse.i16_meld_startindex + 32] := st_drive_cmd.meldungen.sm_halt_axis;
	garr_stoermeldungen[st_config_achse.i16_meld_startindex + 33] := st_drive_cmd.meldungen.sm_motion_command_timeout;
	garr_stoermeldungen[st_config_achse.i16_meld_startindex + 34] := st_sm.b_achsfehler;
	garr_stoermeldungen[st_config_achse.i16_meld_startindex + 35] := st_sm.b_devicefehler;
	garr_stoermeldungen[st_config_achse.i16_meld_startindex + 36] := st_drive_cmd.meldungen.sm_limit_positiv_erreicht;
	garr_stoermeldungen[st_config_achse.i16_meld_startindex + 37] := st_drive_cmd.meldungen.sm_limit_negativ_erreicht;
	garr_stoermeldungen[st_config_achse.i16_meld_startindex + 38] := st_drive_cmd.meldungen.sm_ec_coe_sdo_write_ex;
	garr_stoermeldungen[st_config_achse.i16_meld_startindex + 39] := st_drive_cmd.meldungen.sm_ec_coe_sdo_read_ex;
	garr_stoermeldungen[st_config_achse.i16_meld_startindex + 40] := FALSE;
	garr_stoermeldungen[st_config_achse.i16_meld_startindex + 41] := FALSE;
	garr_stoermeldungen[st_config_achse.i16_meld_startindex + 42] := FALSE;
	garr_stoermeldungen[st_config_achse.i16_meld_startindex + 43] := FALSE;
	garr_stoermeldungen[st_config_achse.i16_meld_startindex + 44] := FALSE;
	garr_stoermeldungen[st_config_achse.i16_meld_startindex + 45] := FALSE;
	garr_stoermeldungen[st_config_achse.i16_meld_startindex + 46] := FALSE;
	garr_stoermeldungen[st_config_achse.i16_meld_startindex + 47] := FALSE;
	garr_stoermeldungen[st_config_achse.i16_meld_startindex + 48] := FALSE;
	garr_stoermeldungen[st_config_achse.i16_meld_startindex + 49] := FALSE;
	garr_stoermeldungen[st_config_achse.i16_meld_startindex + 50] := FALSE;
	garr_stoermeldungen[st_config_achse.i16_meld_startindex + 51] := FALSE;
	garr_stoermeldungen[st_config_achse.i16_meld_startindex + 52] := FALSE;
	garr_stoermeldungen[st_config_achse.i16_meld_startindex + 53] := FALSE;
	garr_stoermeldungen[st_config_achse.i16_meld_startindex + 54] := FALSE;
	garr_stoermeldungen[st_config_achse.i16_meld_startindex + 55] := FALSE;
	garr_stoermeldungen[st_config_achse.i16_meld_startindex + 56] := FALSE;
	garr_stoermeldungen[st_config_achse.i16_meld_startindex + 57] := FALSE;
	garr_stoermeldungen[st_config_achse.i16_meld_startindex + 58] := FALSE;
	garr_stoermeldungen[st_config_achse.i16_meld_startindex + 59] := FALSE;
	garr_stoermeldungen[st_config_achse.i16_meld_startindex + 60] := FALSE;
	garr_stoermeldungen[st_config_achse.i16_meld_startindex + 61] := FALSE;
	garr_stoermeldungen[st_config_achse.i16_meld_startindex + 62] := FALSE;
	garr_stoermeldungen[st_config_achse.i16_meld_startindex + 63] := FALSE;
	garr_stoermeldungen[st_config_achse.i16_meld_startindex + 64] := FALSE;
	garr_stoermeldungen[st_config_achse.i16_meld_startindex + 65] := FALSE;
	garr_stoermeldungen[st_config_achse.i16_meld_startindex + 66] := FALSE;
	garr_stoermeldungen[st_config_achse.i16_meld_startindex + 67] := FALSE;
	garr_stoermeldungen[st_config_achse.i16_meld_startindex + 68] := FALSE;
	garr_stoermeldungen[st_config_achse.i16_meld_startindex + 69] := FALSE;
	garr_stoermeldungen[st_config_achse.i16_meld_startindex + 70] := FALSE;
	garr_stoermeldungen[st_config_achse.i16_meld_startindex + 71] := FALSE;
	garr_stoermeldungen[st_config_achse.i16_meld_startindex + 72] := FALSE;
	garr_stoermeldungen[st_config_achse.i16_meld_startindex + 73] := FALSE;
	garr_stoermeldungen[st_config_achse.i16_meld_startindex + 74] := FALSE;
	garr_stoermeldungen[st_config_achse.i16_meld_startindex + 75] := FALSE;
	garr_stoermeldungen[st_config_achse.i16_meld_startindex + 76] := FALSE;
	garr_stoermeldungen[st_config_achse.i16_meld_startindex + 77] := FALSE;
	garr_stoermeldungen[st_config_achse.i16_meld_startindex + 78] := FALSE;
	garr_stoermeldungen[st_config_achse.i16_meld_startindex + 79] := FALSE;
	garr_stoermeldungen[st_config_achse.i16_meld_startindex + 80] := FALSE;
	garr_stoermeldungen[st_config_achse.i16_meld_startindex + 81] := FALSE;
	garr_stoermeldungen[st_config_achse.i16_meld_startindex + 82] := FALSE;
	garr_stoermeldungen[st_config_achse.i16_meld_startindex + 83] := FALSE;
	garr_stoermeldungen[st_config_achse.i16_meld_startindex + 84] := FALSE;
	garr_stoermeldungen[st_config_achse.i16_meld_startindex + 85] := FALSE;
	garr_stoermeldungen[st_config_achse.i16_meld_startindex + 86] := FALSE;
	garr_stoermeldungen[st_config_achse.i16_meld_startindex + 87] := FALSE;
	garr_stoermeldungen[st_config_achse.i16_meld_startindex + 88] := FALSE;
	garr_stoermeldungen[st_config_achse.i16_meld_startindex + 89] := FALSE;
	garr_stoermeldungen[st_config_achse.i16_meld_startindex + 90] := FALSE;
	garr_stoermeldungen[st_config_achse.i16_meld_startindex + 91] := FALSE;
	garr_stoermeldungen[st_config_achse.i16_meld_startindex + 92] := FALSE;
	garr_stoermeldungen[st_config_achse.i16_meld_startindex + 93] := FALSE;
	garr_stoermeldungen[st_config_achse.i16_meld_startindex + 94] := FALSE;
	garr_stoermeldungen[st_config_achse.i16_meld_startindex + 95] := FALSE;
	garr_stoermeldungen[st_config_achse.i16_meld_startindex + 96] := FALSE;
	garr_stoermeldungen[st_config_achse.i16_meld_startindex + 97] := FALSE;
	garr_stoermeldungen[st_config_achse.i16_meld_startindex + 98] := FALSE;
	garr_stoermeldungen[st_config_achse.i16_meld_startindex + 99] := FALSE;
	
	garr_betriebsmeldungen[st_config_achse.i16_meld_startindex + 0] := FALSE;
	garr_betriebsmeldungen[st_config_achse.i16_meld_startindex + 1] := FALSE;
	garr_betriebsmeldungen[st_config_achse.i16_meld_startindex + 2] := FALSE;
	garr_betriebsmeldungen[st_config_achse.i16_meld_startindex + 3] := FALSE;
	garr_betriebsmeldungen[st_config_achse.i16_meld_startindex + 4] := FALSE;
	garr_betriebsmeldungen[st_config_achse.i16_meld_startindex + 5] := FALSE;
	garr_betriebsmeldungen[st_config_achse.i16_meld_startindex + 6] := FALSE;
	garr_betriebsmeldungen[st_config_achse.i16_meld_startindex + 7] := FALSE;
	garr_betriebsmeldungen[st_config_achse.i16_meld_startindex + 8] := FALSE;
	garr_betriebsmeldungen[st_config_achse.i16_meld_startindex + 9] := FALSE;
	garr_betriebsmeldungen[st_config_achse.i16_meld_startindex + 10] := FALSE;
	garr_betriebsmeldungen[st_config_achse.i16_meld_startindex + 11] := FALSE;
	garr_betriebsmeldungen[st_config_achse.i16_meld_startindex + 12] := FALSE;
	garr_betriebsmeldungen[st_config_achse.i16_meld_startindex + 13] := FALSE;
	garr_betriebsmeldungen[st_config_achse.i16_meld_startindex + 14] := FALSE;
	garr_betriebsmeldungen[st_config_achse.i16_meld_startindex + 15] := FALSE;
	garr_betriebsmeldungen[st_config_achse.i16_meld_startindex + 16] := FALSE;
	garr_betriebsmeldungen[st_config_achse.i16_meld_startindex + 17] := FALSE;
	garr_betriebsmeldungen[st_config_achse.i16_meld_startindex + 18] := FALSE;
	garr_betriebsmeldungen[st_config_achse.i16_meld_startindex + 19] := FALSE;
	garr_betriebsmeldungen[st_config_achse.i16_meld_startindex + 20] := FALSE;
	garr_betriebsmeldungen[st_config_achse.i16_meld_startindex + 21] := FALSE;
	garr_betriebsmeldungen[st_config_achse.i16_meld_startindex + 22] := FALSE;
	garr_betriebsmeldungen[st_config_achse.i16_meld_startindex + 23] := FALSE;
	garr_betriebsmeldungen[st_config_achse.i16_meld_startindex + 24] := FALSE;
	garr_betriebsmeldungen[st_config_achse.i16_meld_startindex + 25] := FALSE;
	garr_betriebsmeldungen[st_config_achse.i16_meld_startindex + 26] := FALSE;
	garr_betriebsmeldungen[st_config_achse.i16_meld_startindex + 27] := FALSE;
	garr_betriebsmeldungen[st_config_achse.i16_meld_startindex + 28] := FALSE;
	garr_betriebsmeldungen[st_config_achse.i16_meld_startindex + 29] := FALSE;
	garr_betriebsmeldungen[st_config_achse.i16_meld_startindex + 30] := FALSE;
	garr_betriebsmeldungen[st_config_achse.i16_meld_startindex + 31] := FALSE;
	garr_betriebsmeldungen[st_config_achse.i16_meld_startindex + 32] := FALSE;
	garr_betriebsmeldungen[st_config_achse.i16_meld_startindex + 33] := FALSE;
	garr_betriebsmeldungen[st_config_achse.i16_meld_startindex + 34] := FALSE;
	garr_betriebsmeldungen[st_config_achse.i16_meld_startindex + 35] := FALSE;
	garr_betriebsmeldungen[st_config_achse.i16_meld_startindex + 36] := FALSE;
	garr_betriebsmeldungen[st_config_achse.i16_meld_startindex + 37] := FALSE;
	garr_betriebsmeldungen[st_config_achse.i16_meld_startindex + 38] := FALSE;
	garr_betriebsmeldungen[st_config_achse.i16_meld_startindex + 39] := FALSE;
	garr_betriebsmeldungen[st_config_achse.i16_meld_startindex + 40] := FALSE;
	garr_betriebsmeldungen[st_config_achse.i16_meld_startindex + 41] := FALSE;
	garr_betriebsmeldungen[st_config_achse.i16_meld_startindex + 42] := FALSE;
	garr_betriebsmeldungen[st_config_achse.i16_meld_startindex + 43] := FALSE;
	garr_betriebsmeldungen[st_config_achse.i16_meld_startindex + 44] := FALSE;
	garr_betriebsmeldungen[st_config_achse.i16_meld_startindex + 45] := FALSE;
	garr_betriebsmeldungen[st_config_achse.i16_meld_startindex + 46] := FALSE;
	garr_betriebsmeldungen[st_config_achse.i16_meld_startindex + 47] := FALSE;
	garr_betriebsmeldungen[st_config_achse.i16_meld_startindex + 48] := FALSE;
	garr_betriebsmeldungen[st_config_achse.i16_meld_startindex + 49] := FALSE;
END_IF
END_PROGRAM

(* POU Rasterfolie/ST_Rasterfolienmontage, ST *)
PROGRAM ST_Rasterfolienmontage
VAR_INPUT
	st_config							: struct_config;
	st_ctrl_in							: struct_ctrl_in;
	b_start_y_Achse					: BOOL;
END_VAR
VAR_IN_OUT
	st_visu							: struct_visu;
END_VAR
VAR_OUTPUT
	st_ctrl_out						: struct_ctrl_out;
END_VAR
VAR
	fb_ton_wz						: TON;
	fb_ton_uez						: TON;
	fb_ton_quitt						: TON;
	fb_r_trig_start						: R_TRIG;
	fb_state_entry						: ST_StateEntry;
	i								: INT := 0;
	arr_rafo_schieberegister			: ARRAY [0..7] OF BOOL;
	sm_keine_rafo_aufgepresst			: BOOL := FALSE;

	e_rasterfolie_aufgepresst			AT %I* : BOOL;
END_VAR
(* Zeiten *)
fb_ton_wz(IN:= , PT:= , Q=>  , ET=> );
fb_ton_uez(IN:= , PT:= t#10s, Q=>  , ET=> );
fb_ton_quitt(IN:= , PT:= t#100ms, Q=> , ET=> );

(* Flanken *)
fb_r_trig_start(CLK:= st_ctrl_in.b_start, Q=> );

(* Toplevel *)
IF fb_state_entry.i16_next_step > INIT AND fb_state_entry.i16_next_step < FEHLER THEN
	IF fb_state_entry.i16_next_step < STOP THEN
		IF st_ctrl_in.b_stop THEN
			fb_state_entry.i16_next_step := STOP;
		END_IF
	END_IF
	(* Allgemeine Fehler *)
	IF zyl_rafo_kamm.st_ctrl.out.b_fehler OR zyl_rafo_vorzentrierer.st_ctrl.out.b_fehler THEN
		fb_state_entry.i16_next_step := FEHLER;

	(* Zylinder im Handbetrieb *)
	ELSIF	gi16_betriebsart = HAND AND
			(st_visu.st_zyl.i16_nr_zyl_im_handbetrieb = zyl_rafo_kamm.fb.st_config.i16_identnummer) OR
			(st_visu.st_zyl.i16_nr_zyl_im_handbetrieb = zyl_rafo_vorzentrierer.fb.st_config.i16_identnummer)
			THEN
				fb_state_entry.i16_next_step := FEHLER;
	END_IF
END_IF

(* ======================================Schrittkette======================================== *)
fb_state_entry(
	i16_next_step:= ,
	i16_pos:= 1,
	s_debugtext:= ,
	E=> ,
	X=> ,
	i16_step=> ,
	i16_last_step=> );

CASE fb_state_entry.i16_step OF
(*=======================================================*)
	INIT_OBJ:
		IF st_config.b_config_fertig THEN
			fb_state_entry.i16_next_step := INIT;
		END_IF

(*=======================================================*)
	INIT:
		IF fb_state_entry.E THEN
			fb_ton_wz.IN := FALSE;
			fb_ton_uez.IN := FALSE;
			fb_ton_quitt.IN := FALSE;
			st_ctrl_out.b_fehler := FALSE;
			st_ctrl_out.b_bereit := FALSE;
			st_ctrl_out.b_fertig := FALSE;
			st_ctrl_out.b_fertig_2 := FALSE;
			zyl_rafo_kamm.st_ctrl.in.b_ausfahren := FALSE;
			zyl_rafo_kamm.st_ctrl.in.b_einfahren := FALSE;
			zyl_rafo_vorzentrierer.st_ctrl.in.b_ausfahren := FALSE;
			zyl_rafo_vorzentrierer.st_ctrl.in.b_einfahren := FALSE;
			rasterfolieneinzug.st_ctrl.in.b_start := FALSE;
			sm_keine_rafo_aufgepresst := FALSE;

			FOR i := 0 TO 7 BY 1 DO
				arr_rafo_schieberegister[i] := FALSE;
			END_FOR
		END_IF

		(*-----------------------Weiterschaltbedingungen----------------------------*)
		IF st_ctrl_in.b_init THEN
			zyl_rafo_kamm.st_ctrl.in.b_quittieren := FALSE;
			fb_state_entry.i16_next_step := 20;
		END_IF

(*=======================================================*)
	20:	(* Kamm einfahren *)
		IF fb_state_entry.E THEN
			zyl_rafo_kamm.st_ctrl.in.b_ausfahren := TRUE;
		END_IF

		(*-----------------------Weiterschaltbedingungen----------------------------*)
		IF zyl_rafo_kamm.st_ctrl.out.b_ausgefahren  THEN
			zyl_rafo_kamm.st_ctrl.in.b_ausfahren := FALSE;
			IF gst_datensatz.st_wkz.b_rafo_vorzentrierer_aktiv THEN
				fb_state_entry.i16_next_step := 30;
			ELSE
				fb_state_entry.i16_next_step := BEREIT;
			END_IF
		END_IF

(*=======================================================*)
	30:	(* Vorzentrierer einfahren *)
		IF fb_state_entry.E THEN
			zyl_rafo_vorzentrierer.st_ctrl.in.b_ausfahren := TRUE;	(*Federrückstellung*)
		END_IF

		(*-----------------------Weiterschaltbedingungen----------------------------*)
		IF  zyl_rafo_vorzentrierer.st_ctrl.out.b_ausgefahren THEN
			zyl_rafo_vorzentrierer.st_ctrl.in.b_ausfahren := FALSE;
			fb_state_entry.i16_next_step := BEREIT;
		END_IF

(*=======================================================*)
	BEREIT:
		IF fb_state_entry.E THEN
			st_ctrl_out.b_bereit := TRUE;
			st_ctrl_out.b_fertig := TRUE;
			st_ctrl_out.b_fertig_2 := TRUE;
		END_IF

		(*-----------------------Weiterschaltbedingungen----------------------------*)
		IF st_ctrl_in.b_start THEN
			st_ctrl_out.b_fertig := FALSE;
			st_ctrl_out.b_fertig_2 := FALSE;
			b_start_y_Achse := FALSE;
			fb_state_entry.i16_next_step := 110;
		END_IF

(*=======================================================*)
	110: (* Positioniere Achse wieder zurück auf  0-Koordinate  des ISK *)
		IF fb_state_entry.E THEN
			ST_Y_Achse.lr_tmp_Achspos:=
							gst_datensatz.st_isk.lr_pos_y_0 +
							gst_datensatz.st_wkz.lr_offset_y_pos_0 +
							gst_datensatz.st_wt.lr_offset_y_pos_0 +
							gst_datensatz.st_md.lr_offset_y_pos_0 +
							gst_datensatz.st_bestueckprogramm.lr_y[0];
			b_start_y_Achse := TRUE;
		END_IF

		(*-----------------------Weiterschaltbedingungen----------------------------*)
		IF 	ST_Y_Achse.st_drive_cmd.enu_cmd = NO_COMMAND AND
			NOT b_start_y_Achse THEN
			fb_state_entry.i16_next_step := 117;
		END_IF

(*=======================================================*)
	117:	(* Vorzentrierung vorhanden *)

	IF gst_datensatz.st_wkz.b_rafo_vorzentrierer_aktiv THEN
		fb_state_entry.i16_next_step := 118;
	ELSE
		fb_state_entry.i16_next_step :=120;
	END_IF

(*=======================================================*)
	118:	(* Vorzentrierung ausfahren *)
		IF fb_state_entry.E THEN
			zyl_rafo_vorzentrierer.st_ctrl.in.b_einfahren := TRUE;		(*Nicht Federrückstellend*)
		END_IF

		(*-----------------------Weiterschaltbedingungen----------------------------*)
		IF zyl_rafo_vorzentrierer.st_ctrl.out.b_eingefahren AND gb_ba_auto_kontroller THEN
			zyl_rafo_vorzentrierer.st_ctrl.in.b_einfahren := FALSE;
			fb_state_entry.i16_next_step := 120;
		END_IF

(*=======================================================*)
	120:	(* Kamm zum Gegenhalten ausfahren *)
		IF fb_state_entry.E THEN
			zyl_rafo_kamm.st_ctrl.in.b_einfahren := TRUE;
		END_IF

		(*-----------------------Weiterschaltbedingungen----------------------------*)
		IF zyl_rafo_kamm.st_ctrl.out.b_eingefahren AND gb_ba_auto_kontroller THEN
			zyl_rafo_kamm.st_ctrl.in.b_einfahren := FALSE;
			fb_state_entry.i16_next_step := 130;
		END_IF

(*=======================================================*)
	130: (* Warte *)
		IF fb_state_entry.E THEN
			fb_ton_wz.PT := t#100ms;
 			fb_ton_wz.IN := TRUE;
		END_IF

		(*-----------------------Weiterschaltbedingungen----------------------------*)
		IF fb_ton_wz.Q THEN
			fb_ton_wz.IN := FALSE;
			fb_state_entry.i16_next_step := 140;
		END_IF

(*=======================================================*)
	140:	(* Y-Achse muss runter fahren auf Absenkposition *)

		IF fb_state_entry.E THEN
			ST_Y_Achse.lr_tmp_Achspos:=	gst_datensatz.st_wkz.st_rasterfolie.lr_pos_absenken
											+ gst_datensatz.st_md.lr_offset_y_pos_0;
			b_start_y_Achse := TRUE;
		END_IF

		(*-----------------------Weiterschaltbedingungen----------------------------*)
		IF ST_Y_Achse.st_drive_cmd.enu_cmd = NO_COMMAND AND
			NOT b_start_y_Achse THEN
			fb_state_entry.i16_next_step := 150;
		END_IF

(*=======================================================*)
	150:	(* Eine Rasterfolie mit der Bestückachse setzen *)
		IF fb_state_entry.E THEN
			axis_virt_master.st_ctrl.in.b_start := TRUE;
		END_IF

		(*-----------------------Weiterschaltbedingungen----------------------------*)
		IF  axis_virt_master.st_ctrl.out.b_fertig AND NOT fb_state_entry.E AND gb_ba_auto_kontroller THEN
			axis_virt_master.st_ctrl.in.b_start := FALSE;
			fb_state_entry.i16_next_step := 160;
		END_IF

(*=======================================================*)
	160: (* Warte bis Y-Achse wieder hoch gefahren ist auf  0-Koordinate  des ISK *)

		IF fb_state_entry.E THEN
			ST_Y_Achse.lr_tmp_Achspos:=
							gst_datensatz.st_isk.lr_pos_y_0 +
							gst_datensatz.st_wkz.lr_offset_y_pos_0 +
							gst_datensatz.st_wt.lr_offset_y_pos_0 +
							gst_datensatz.st_md.lr_offset_y_pos_0 +
							gst_datensatz.st_bestueckprogramm.lr_y[0];
			b_start_y_Achse := TRUE;
		END_IF

		(*-----------------------Weiterschaltbedingungen----------------------------*)
		IF ST_Y_Achse.st_drive_cmd.enu_cmd = NO_COMMAND AND
			NOT b_start_y_Achse THEN
			fb_state_entry.i16_next_step := 170;
		END_IF

(*=======================================================*)
	170: (* Warte *)
		IF fb_state_entry.E THEN
			fb_ton_wz.PT := t#100ms;
 			fb_ton_wz.IN := TRUE;
		END_IF

		(*-----------------------Weiterschaltbedingungen----------------------------*)
		IF fb_ton_wz.Q THEN
			fb_ton_wz.IN := FALSE;
			fb_state_entry.i16_next_step := 180;
		END_IF

(*=======================================================*)
	180:	(* Kamm einfahren *)
		IF fb_state_entry.E THEN
			zyl_rafo_kamm.st_ctrl.in.b_ausfahren := TRUE;
			IF gst_datensatz.st_wkz.b_rafo_vorzentrierer_aktiv THEN
				zyl_rafo_vorzentrierer.st_ctrl.in.b_ausfahren := TRUE;	(*Federrückstellung*)
			END_IF
		END_IF

		(*-----------------------Weiterschaltbedingungen----------------------------*)
		IF gst_datensatz.st_wkz.b_rafo_vorzentrierer_aktiv
			AND zyl_rafo_kamm.st_ctrl.out.b_ausgefahren AND zyl_rafo_vorzentrierer.st_ctrl.out.b_ausgefahren
				AND gb_ba_auto_kontroller THEN
					zyl_rafo_kamm.st_ctrl.in.b_ausfahren := FALSE;
					zyl_rafo_vorzentrierer.st_ctrl.in.b_ausfahren := FALSE;
				fb_state_entry.i16_next_step := 185;
		ELSIF NOT gst_datensatz.st_wkz.b_rafo_vorzentrierer_aktiv AND  zyl_rafo_kamm.st_ctrl.out.b_ausgefahren
				AND gb_ba_auto_kontroller THEN
					zyl_rafo_kamm.st_ctrl.in.b_ausfahren := FALSE;
				fb_state_entry.i16_next_step := 185;
		END_IF

(*=======================================================*)
	185: (* Warte bis Y-Achse wieder runter gefahren ist (auf Einfahrhöhe) *)
		IF fb_state_entry.E THEN
			ST_Y_Achse.lr_tmp_Achspos:= gst_datensatz.st_wkz.st_yz_tisch.r_wkz_einfahrpos_y;
			b_start_y_Achse := TRUE;
		END_IF

		(*-----------------------Weiterschaltbedingungen----------------------------*)
		IF ST_Y_Achse.st_drive_cmd.enu_cmd = NO_COMMAND AND
			NOT b_start_y_Achse THEN
			st_ctrl_out.b_fertig := TRUE;
			fb_state_entry.i16_next_step := 190;
		END_IF
(*=======================================================*)
	190:
		IF	ST_Z_Achse.st_drive_cmd.enu_cmd = MOVE_ABSOLUTE THEN
			fb_state_entry.i16_next_step := 200;
		END_IF

(*=======================================================*)
	200: (* Warte bis Z-Achse zwischen die GLS fährt zur Überprüfung der Rasterfolie auf dem STV *)
		IF fb_state_entry.E THEN
			arr_rafo_schieberegister[ST_Z_Achse.i32_anzahl_rasterfolie] := FALSE;
			fb_ton_uez.IN:=FALSE;
		END_IF

		(*-----------------------Weiterschaltbedingungen----------------------------*)
			(* Überprüfung GLS-Signal *)
		IF	ST_Z_Achse.st_drive_cmd.enu_cmd = NO_COMMAND THEN
			fb_ton_uez(IN:=TRUE,PT:=t#4s);
			IF e_rasterfolie_aufgepresst  THEN
				(* Rasterfolie vorhanden *)
				arr_rafo_schieberegister[ST_Z_Achse.i32_anzahl_rasterfolie] := TRUE;
				fb_state_entry.i16_next_step := BEREIT;
			ELSIF fb_ton_uez.Q THEN
				(* Keine Rasterfolie auf dem STV *)
				sm_keine_rafo_aufgepresst := TRUE;
				fb_state_entry.i16_next_step := FEHLER;
			END_IF
		END_IF

		IF fb_state_entry.X THEN
			fb_ton_uez.IN:=FALSE;
		END_IF

(*=======================================================*)
	FEHLER:
		IF fb_state_entry.E THEN
			st_ctrl_out.b_fehler := TRUE;
			fb_ton_quitt.IN := FALSE;
			zyl_rafo_kamm.st_ctrl.in.b_quittieren := FALSE;
			zyl_rafo_vorzentrierer.st_ctrl.in.b_quittieren := FALSE;
		END_IF

		(*-----------------------Weiterschaltbedingungen----------------------------*)
		IF st_ctrl_in.b_quitt AND NOT fb_state_entry.E THEN
			st_ctrl_out.b_fehler := FALSE;
			zyl_rafo_kamm.st_ctrl.in.b_quittieren := TRUE;
			zyl_rafo_vorzentrierer.st_ctrl.in.b_quittieren := TRUE;
			fb_ton_quitt.IN := TRUE;
		END_IF

		IF fb_ton_quitt.Q THEN
			fb_ton_quitt.IN := FALSE;
			fb_state_entry.i16_next_step := INIT;
		END_IF

(*=======================================================*)
	STOP:
		IF fb_state_entry.E THEN
			fb_ton_quitt.IN := FALSE;
			zyl_rafo_kamm.st_ctrl.in.b_quittieren := FALSE;
			zyl_rafo_vorzentrierer.st_ctrl.in.b_quittieren := FALSE;
		END_IF

		(*-----------------------Weiterschaltbedingungen----------------------------*)
		IF st_ctrl_in.b_quitt AND NOT fb_state_entry.E THEN
			fb_ton_quitt.IN := TRUE;
			zyl_rafo_kamm.st_ctrl.in.b_quittieren := TRUE;
			zyl_rafo_vorzentrierer.st_ctrl.in.b_quittieren := TRUE;
		END_IF

		IF fb_ton_quitt.Q THEN
			fb_ton_quitt.IN := FALSE;
			fb_state_entry.i16_next_step := INIT;
		END_IF
END_CASE

fb_state_entry(
	i16_next_step:= , 
	i16_pos:= 2,
	s_debugtext:= ,
	E=> , 
	X=> , 
	i16_step=> ,
	i16_last_step=> );

IF st_config.b_config_fertig THEN
	(* Fehlermeldungen und Betriebsmeldungen ab dem Startindex in die globalen Meldungsarrays schreiben *)
	garr_stoermeldungen[st_config.i16_meld_startindex + 0] := sm_keine_rafo_aufgepresst;
	garr_stoermeldungen[st_config.i16_meld_startindex + 1] := FALSE;
	garr_stoermeldungen[st_config.i16_meld_startindex + 2] := FALSE;
	garr_stoermeldungen[st_config.i16_meld_startindex + 3] := FALSE;
	garr_stoermeldungen[st_config.i16_meld_startindex + 4] := FALSE;
	garr_stoermeldungen[st_config.i16_meld_startindex + 5] := FALSE;
	garr_stoermeldungen[st_config.i16_meld_startindex + 6] := FALSE;
	garr_stoermeldungen[st_config.i16_meld_startindex + 7] := FALSE;
	garr_stoermeldungen[st_config.i16_meld_startindex + 8] := FALSE;
	garr_stoermeldungen[st_config.i16_meld_startindex + 9] := FALSE;
	garr_stoermeldungen[st_config.i16_meld_startindex + 10] := FALSE;
	garr_stoermeldungen[st_config.i16_meld_startindex + 11] := FALSE;
	garr_stoermeldungen[st_config.i16_meld_startindex + 12] := FALSE;
	garr_stoermeldungen[st_config.i16_meld_startindex + 13] := FALSE;
	garr_stoermeldungen[st_config.i16_meld_startindex + 14] := FALSE;
	garr_stoermeldungen[st_config.i16_meld_startindex + 15] := FALSE;
	garr_stoermeldungen[st_config.i16_meld_startindex + 16] := FALSE;
	garr_stoermeldungen[st_config.i16_meld_startindex + 17] := FALSE;
	garr_stoermeldungen[st_config.i16_meld_startindex + 18] := FALSE;
	garr_stoermeldungen[st_config.i16_meld_startindex + 19] := FALSE;
	
	garr_betriebsmeldungen[st_config.i16_meld_startindex + 0] := FALSE;
	garr_betriebsmeldungen[st_config.i16_meld_startindex + 1] := FALSE;
	garr_betriebsmeldungen[st_config.i16_meld_startindex + 2] := FALSE;
	garr_betriebsmeldungen[st_config.i16_meld_startindex + 3] := FALSE;
	garr_betriebsmeldungen[st_config.i16_meld_startindex + 4] := FALSE;
	garr_betriebsmeldungen[st_config.i16_meld_startindex + 5] := FALSE;
	garr_betriebsmeldungen[st_config.i16_meld_startindex + 6] := FALSE;
	garr_betriebsmeldungen[st_config.i16_meld_startindex + 7] := FALSE;
	garr_betriebsmeldungen[st_config.i16_meld_startindex + 8] := FALSE;
	garr_betriebsmeldungen[st_config.i16_meld_startindex + 9] := FALSE;
	garr_betriebsmeldungen[st_config.i16_meld_startindex + 10] := FALSE;
	garr_betriebsmeldungen[st_config.i16_meld_startindex + 11] := FALSE;
	garr_betriebsmeldungen[st_config.i16_meld_startindex + 12] := FALSE;
	garr_betriebsmeldungen[st_config.i16_meld_startindex + 13] := FALSE;
	garr_betriebsmeldungen[st_config.i16_meld_startindex + 14] := FALSE;
	garr_betriebsmeldungen[st_config.i16_meld_startindex + 15] := FALSE;
	garr_betriebsmeldungen[st_config.i16_meld_startindex + 16] := FALSE;
	garr_betriebsmeldungen[st_config.i16_meld_startindex + 17] := FALSE;
	garr_betriebsmeldungen[st_config.i16_meld_startindex + 18] := FALSE;
	garr_betriebsmeldungen[st_config.i16_meld_startindex + 19] := FALSE;
END_IF
END_PROGRAM

(* POU Rasterfolie/ST_Rasterfolieneinzug, ST *)
PROGRAM ST_Rasterfolieneinzug
VAR_INPUT
	st_config							: struct_config;
	st_ctrl_in							: struct_ctrl_in;
END_VAR
VAR_IN_OUT
	st_visu							: struct_visu;
END_VAR
VAR_OUTPUT
	st_ctrl_out						: struct_ctrl_out;
END_VAR
VAR
	fb_ton_wz						: TON;
	fb_ton_uez						: TON;
	fb_ton_quitt						: TON;
	fb_ton_gls_rafo_vorhanden		: TON;
	fb_tof_gls_rafo_ende			: TOF;
	fb_tof_AbschaltungIonisierung		: TOF;
	fb_r_trig_start						: R_TRIG;
	fb_r_trig_vorschubkontrolle			: R_TRIG;
	fb_f_trig_vorschubkontrolle			: F_TRIG;
	fb_state_entry						: ST_StateEntry;
	i								: INT := 0;
	sm_fehler_rafo_vorschub			: BOOL := FALSE;
	sm_keine_rafo_im_einzug		: BOOL := FALSE;

	e_rasfo_ende						AT %I* : BOOL;
	e_rasfo_vorschubkontrolle			AT %I* : BOOL;
	e_rasfo_rueckzugueberwachung		AT %I* : BOOL;

	(* Ausgang Ionisierung Rasterfolie einschalten *)
	aIonisierungEin				AT %Q* : BOOL;

END_VAR
(* Zeiten *)
fb_ton_wz(IN:= , PT:= , Q=>  , ET=> );
fb_ton_uez(IN:= , PT:= t#1000ms, Q=>  , ET=> );
fb_ton_quitt(IN:= , PT:= t#100ms, Q=> , ET=> );
fb_ton_gls_rafo_vorhanden(IN:= e_rasfo_ende, PT:= T#300ms, Q=> , ET=> );
fb_tof_gls_rafo_ende(IN:= fb_ton_gls_rafo_vorhanden.Q, PT:= T#300ms, Q=> , ET=> );
fb_tof_AbschaltungIonisierung(IN:= fb_state_entry.i16_step = 200, PT:= T#2m, Q=> , ET=> );

(* Flanken *)
fb_r_trig_start(CLK:= st_ctrl_in.b_start, Q=> );
fb_r_trig_vorschubkontrolle(CLK:= e_rasfo_vorschubkontrolle, Q=> );
fb_f_trig_vorschubkontrolle(CLK:= e_rasfo_vorschubkontrolle, Q=> );


(* Steuerung Ionisierung *)
IF gi16_maschinenstatusinfo = STATUS_MASCHINE_ARBEITET THEN
	aIonisierungEin := fb_tof_AbschaltungIonisierung.Q;
ELSE
	aIonisierungEin := FALSE;
END_IF


(* Toplevel *)
IF fb_state_entry.i16_next_step > INIT AND fb_state_entry.i16_next_step < FEHLER THEN
	IF fb_state_entry.i16_next_step < STOP THEN
		IF st_ctrl_in.b_stop THEN
			fb_state_entry.i16_next_step := STOP;
		END_IF
	END_IF
	(* Allgemeine Fehler *)
	IF	zyl_rafo_faenger.st_ctrl.out.b_fehler OR
		zyl_rafo_klemmen.st_ctrl.out.b_fehler OR
		zyl_rafo_vorschub.st_ctrl.out.b_fehler
		THEN
			fb_state_entry.i16_next_step := FEHLER;

	(* Zylinder im Handbetrieb *)
	ELSIF	gi16_betriebsart = HAND AND (
			(st_visu.st_zyl.i16_nr_zyl_im_handbetrieb = zyl_rafo_faenger.fb.st_config.i16_identnummer) OR
			(st_visu.st_zyl.i16_nr_zyl_im_handbetrieb = zyl_rafo_klemmen.fb.st_config.i16_identnummer) OR
			(st_visu.st_zyl.i16_nr_zyl_im_handbetrieb = zyl_rafo_vorschub.fb.st_config.i16_identnummer) )
			THEN
				fb_state_entry.i16_next_step := FEHLER;
	END_IF
END_IF

sm_keine_rafo_im_einzug:=ST_Z_Achse.sm_keine_rafo_im_einzug;

(* ======================================Schrittkette======================================== *)
fb_state_entry(
	i16_next_step:= ,
	i16_pos:= 1,
	s_debugtext:= ,
	E=> ,
	X=> , 
	i16_step=> ,
	i16_last_step=> );

CASE fb_state_entry.i16_step OF
(*=======================================================*)
	INIT_OBJ:
		IF st_config.b_config_fertig THEN
			fb_state_entry.i16_next_step := INIT;
		END_IF

(*=======================================================*)
	INIT:
		IF fb_state_entry.E THEN
			fb_ton_wz.IN := FALSE;
			fb_ton_uez.IN := FALSE;
			fb_ton_quitt.IN := FALSE;
			st_ctrl_out.b_fehler := FALSE;
			st_ctrl_out.b_bereit := FALSE;
			st_ctrl_out.b_fertig := FALSE;
			zyl_rafo_faenger.st_ctrl.in.b_ausfahren := FALSE;
			zyl_rafo_faenger.st_ctrl.in.b_einfahren := FALSE;
			zyl_rafo_klemmen.st_ctrl.in.b_ausfahren := FALSE;
			zyl_rafo_klemmen.st_ctrl.in.b_einfahren := FALSE;
			zyl_rafo_vorschub.st_ctrl.in.b_ausfahren := FALSE;
			zyl_rafo_vorschub.st_ctrl.in.b_einfahren := FALSE;
			sm_fehler_rafo_vorschub := FALSE;
			sm_keine_rafo_im_einzug := FALSE;
		END_IF

		(*-----------------------Weiterschaltbedingungen----------------------------*)
		IF st_ctrl_in.b_init THEN
			zyl_rafo_faenger.st_ctrl.in.b_quittieren := FALSE;
			zyl_rafo_klemmen.st_ctrl.in.b_quittieren := FALSE;
			zyl_rafo_vorschub.st_ctrl.in.b_quittieren := FALSE;
			IF gst_datensatz.st_md.b_wt_transport_simulation THEN
				fb_state_entry.i16_next_step := BEREIT;
			ELSE
				fb_state_entry.i16_next_step := 20;
			END_IF
		END_IF

(*=======================================================*)
	20:	(* Klemmung ausfahren und Folie halten *)
		IF fb_state_entry.E THEN
			zyl_rafo_klemmen.st_ctrl.in.b_ausfahren := TRUE;
		END_IF

		(*-----------------------Weiterschaltbedingungen----------------------------*)
		IF zyl_rafo_klemmen.st_ctrl.out.b_ausgefahren THEN
			zyl_rafo_klemmen.st_ctrl.in.b_ausfahren := FALSE;
			fb_state_entry.i16_next_step := 30;
		END_IF

(*=======================================================*)
	30:	(* Fänger einfahren *)
		IF fb_state_entry.E THEN
			zyl_rafo_faenger.st_ctrl.in.b_einfahren := TRUE;
		END_IF

		(*-----------------------Weiterschaltbedingungen----------------------------*)
		IF zyl_rafo_faenger.st_ctrl.out.b_eingefahren THEN
			zyl_rafo_faenger.st_ctrl.in.b_einfahren := FALSE;
			fb_state_entry.i16_next_step := 40;
		END_IF

(*=======================================================*)
	40:	(* Vorschub zurück fahren *)
		IF fb_state_entry.E THEN
			zyl_rafo_vorschub.st_ctrl.in.b_einfahren := TRUE;
		END_IF

		(*-----------------------Weiterschaltbedingungen----------------------------*)
		IF zyl_rafo_vorschub.st_ctrl.out.b_eingefahren THEN
			zyl_rafo_vorschub.st_ctrl.in.b_einfahren := FALSE;
			fb_state_entry.i16_next_step := 50;
		END_IF

(*=======================================================*)
	50:	(* Fänger ausfahren *)
		IF fb_state_entry.E THEN
			zyl_rafo_faenger.st_ctrl.in.b_ausfahren := TRUE;
		END_IF

		(*-----------------------Weiterschaltbedingungen----------------------------*)
		IF zyl_rafo_faenger.st_ctrl.out.b_ausgefahren THEN
			zyl_rafo_faenger.st_ctrl.in.b_ausfahren := FALSE;
			fb_state_entry.i16_next_step := 60;
		END_IF

(*=======================================================*)
	60:	(* Klemmung einfahren *)
		IF fb_state_entry.E THEN
			zyl_rafo_klemmen.st_ctrl.in.b_einfahren := TRUE;
		END_IF

		(*-----------------------Weiterschaltbedingungen----------------------------*)
		IF zyl_rafo_klemmen.st_ctrl.out.b_eingefahren THEN
			zyl_rafo_klemmen.st_ctrl.in.b_einfahren := FALSE;
			fb_state_entry.i16_next_step := BEREIT;
		END_IF

(*=======================================================*)
	BEREIT:
		IF fb_state_entry.E THEN
			st_ctrl_out.b_bereit := TRUE;
			st_ctrl_out.b_fertig := TRUE;
		END_IF

		(*-----------------------Weiterschaltbedingungen----------------------------*)
		IF st_ctrl_in.b_start THEN
			st_ctrl_out.b_fertig := FALSE;
			fb_state_entry.i16_next_step := 110;
		END_IF

(*=======================================================*)
	110:	(* Prüfe Rasterfolie im Einzug *)		(*wird im BEREIT der Z-Achse geprütf*)

		fb_state_entry.i16_next_step := 200;

(*===========================Vorschub Folie============================*)
	200:	(* Vorschub ausfahren und Vorschub prüfen *)
		IF fb_state_entry.E THEN
			zyl_rafo_vorschub.st_ctrl.in.b_ausfahren := TRUE;
		END_IF

		(*-----------------------Weiterschaltbedingungen----------------------------*)
		(* Vorschubkontrolle durch positive Flanke *)
		IF fb_r_trig_vorschubkontrolle.Q THEN
			fb_state_entry.i16_next_step := 210;
		ELSIF zyl_rafo_vorschub.st_ctrl.out.b_ausgefahren THEN
			sm_fehler_rafo_vorschub := TRUE;
			fb_state_entry.i16_next_step := FEHLER;
		END_IF

(*=======================================================*)
	210:	(* Verhindere Signalüberschneidungen *)
		IF fb_state_entry.E THEN
			fb_ton_wz.PT := t#1000ms;
 			fb_ton_wz.IN := TRUE;
		END_IF

		(*-----------------------Weiterschaltbedingungen----------------------------*)
		(* Vorschubkontrolle durch negative Flanke *)
		IF fb_f_trig_vorschubkontrolle.Q THEN
			fb_ton_wz.IN := FALSE;
			fb_state_entry.i16_next_step := 220;
		ELSIF zyl_rafo_vorschub.st_ctrl.out.b_ausgefahren AND fb_ton_wz.Q THEN
			sm_fehler_rafo_vorschub := TRUE;
			fb_state_entry.i16_next_step := FEHLER;
		END_IF

(*=======================================================*)
	220:	(* Vorschub ist fertig ausgefahren *)

		(*-----------------------Weiterschaltbedingungen----------------------------*)
		IF zyl_rafo_vorschub.st_ctrl.out.b_ausgefahren AND gb_ba_auto_kontroller THEN
			zyl_rafo_vorschub.st_ctrl.in.b_ausfahren := FALSE;
			fb_state_entry.i16_next_step := 230;
		END_IF

(*=======================================================*)
	230:	(* Klemmung ausfahren und Folie halten *)
		IF fb_state_entry.E THEN
			zyl_rafo_klemmen.st_ctrl.in.b_ausfahren := TRUE;
		END_IF

		(*-----------------------Weiterschaltbedingungen----------------------------*)
		IF zyl_rafo_klemmen.st_ctrl.out.b_ausgefahren AND gb_ba_auto_kontroller THEN
			zyl_rafo_klemmen.st_ctrl.in.b_ausfahren := FALSE;
			fb_state_entry.i16_next_step := 240;
		END_IF

(*=======================================================*)
	240:	(* Fänger einfahren *)
		IF fb_state_entry.E THEN
			zyl_rafo_faenger.st_ctrl.in.b_einfahren := TRUE;
		END_IF

		(*-----------------------Weiterschaltbedingungen----------------------------*)
		IF zyl_rafo_faenger.st_ctrl.out.b_eingefahren AND gb_ba_auto_kontroller THEN
			zyl_rafo_faenger.st_ctrl.in.b_einfahren := FALSE;
			fb_state_entry.i16_next_step := 250;
		END_IF

(*=======================================================*)
	250:	(* Vorschub zurück fahren *)
		IF fb_state_entry.E THEN
			zyl_rafo_vorschub.st_ctrl.in.b_einfahren := TRUE;
		END_IF

		(*-----------------------Weiterschaltbedingungen----------------------------*)
		IF zyl_rafo_vorschub.st_ctrl.out.b_eingefahren AND gb_ba_auto_kontroller THEN
			zyl_rafo_vorschub.st_ctrl.in.b_einfahren := FALSE;
			fb_state_entry.i16_next_step := 260;
		END_IF

(*=======================================================*)
	260: (* Warte *)
		IF fb_state_entry.E THEN
			fb_ton_wz.PT := t#300ms;
 			fb_ton_wz.IN := TRUE;
		END_IF

		(*-----------------------Weiterschaltbedingungen----------------------------*)
		IF fb_ton_wz.Q THEN
			fb_ton_wz.IN := FALSE;
			(* Rasterfolieneinzug lüften
			Dies wird nur gemacht, wenn die Nocken ungleich 0 sind und Anfangs- und Endnocke aunterschiedlich sind
			Zwischen den Nocken wird die Rasterfolie vom Werkzeug gehalten *)
			IF gst_datensatz.st_wkz.nockenschaltwerk_bestueckachse.arr_nocken[NO_RASTERFOLIE_LUEFTEN].r_cam_begin <> 0 AND
				gst_datensatz.st_wkz.nockenschaltwerk_bestueckachse.arr_nocken[NO_RASTERFOLIE_LUEFTEN].r_cam_begin <> gst_datensatz.st_wkz.nockenschaltwerk_bestueckachse.arr_nocken[NO_RASTERFOLIE_LUEFTEN].r_cam_end THEN
				fb_state_entry.i16_next_step := 290;(* Ablauf mit Lüften *)
			ELSE
				fb_state_entry.i16_next_step := 270;(* Ablauf ohne Lüften *)
			END_IF
		END_IF

(*=======================================================*)
	270:	(* Fänger ausfahren *)
		IF fb_state_entry.E THEN
			zyl_rafo_faenger.st_ctrl.in.b_ausfahren := TRUE;
		END_IF

		(*-----------------------Weiterschaltbedingungen----------------------------*)
		IF zyl_rafo_faenger.st_ctrl.out.b_ausgefahren AND gb_ba_auto_kontroller THEN
			zyl_rafo_faenger.st_ctrl.in.b_ausfahren := FALSE;
			fb_state_entry.i16_next_step := 280;
		END_IF

(*=======================================================*)
	280:	(* Klemmung einfahren *)
		IF fb_state_entry.E THEN
			zyl_rafo_klemmen.st_ctrl.in.b_einfahren := TRUE;
		END_IF

		(*-----------------------Weiterschaltbedingungen----------------------------*)
		IF zyl_rafo_klemmen.st_ctrl.out.b_eingefahren AND gb_ba_auto_kontroller THEN
			zyl_rafo_klemmen.st_ctrl.in.b_einfahren := FALSE;
			fb_state_entry.i16_next_step := 290;
		END_IF

(*=======================================================*)
	290:	(* Bandüberstand nach WKZ prüfen und eventuell zurückziehen *)

		(*-----------------------Weiterschaltbedingungen----------------------------*)
		IF e_rasfo_rueckzugueberwachung THEN
			fb_state_entry.i16_next_step := 300;
		ELSE
			fb_state_entry.i16_next_step := BEREIT;
		END_IF

(*===========================Rückzug Folie============================*)
	300:	(* Klemmung ausfahren und Folie halten *)
		IF fb_state_entry.E THEN
			zyl_rafo_klemmen.st_ctrl.in.b_ausfahren := TRUE;
		END_IF

		(*-----------------------Weiterschaltbedingungen----------------------------*)
		IF zyl_rafo_klemmen.st_ctrl.out.b_ausgefahren AND gb_ba_auto_kontroller THEN
			zyl_rafo_klemmen.st_ctrl.in.b_ausfahren := FALSE;
			fb_state_entry.i16_next_step := 310;
		END_IF

(*=======================================================*)
	310:	(* Fänger einfahren *)
		IF fb_state_entry.E THEN
			zyl_rafo_faenger.st_ctrl.in.b_einfahren := TRUE;
		END_IF

		(*-----------------------Weiterschaltbedingungen----------------------------*)
		IF zyl_rafo_faenger.st_ctrl.out.b_eingefahren AND gb_ba_auto_kontroller THEN
			zyl_rafo_faenger.st_ctrl.in.b_einfahren := FALSE;
			fb_state_entry.i16_next_step := 320;
		END_IF

(*=======================================================*)
	320:	(* Vorschub ausfahren *)
		IF fb_state_entry.E THEN
			zyl_rafo_vorschub.st_ctrl.in.b_ausfahren := TRUE;
		END_IF

		(*-----------------------Weiterschaltbedingungen----------------------------*)
		IF zyl_rafo_vorschub.st_ctrl.out.b_ausgefahren AND gb_ba_auto_kontroller THEN
			zyl_rafo_vorschub.st_ctrl.in.b_ausfahren := FALSE;
			fb_state_entry.i16_next_step := 330;
		END_IF

(*=======================================================*)
	330:	(* Fänger ausfahren *)
		IF fb_state_entry.E THEN
			zyl_rafo_faenger.st_ctrl.in.b_ausfahren := TRUE;
		END_IF

		(*-----------------------Weiterschaltbedingungen----------------------------*)
		IF zyl_rafo_faenger.st_ctrl.out.b_ausgefahren AND gb_ba_auto_kontroller THEN
			zyl_rafo_faenger.st_ctrl.in.b_ausfahren := FALSE;
			fb_state_entry.i16_next_step := 340;
		END_IF

(*=======================================================*)
	340:	(* Klemmung einfahren *)
		IF fb_state_entry.E THEN
			zyl_rafo_klemmen.st_ctrl.in.b_einfahren := TRUE;
		END_IF

		(*-----------------------Weiterschaltbedingungen----------------------------*)
		IF zyl_rafo_klemmen.st_ctrl.out.b_eingefahren AND gb_ba_auto_kontroller THEN
			zyl_rafo_klemmen.st_ctrl.in.b_einfahren := FALSE;
			fb_state_entry.i16_next_step := 350;
		END_IF

(*=======================================================*)
	350:	(* Vorschub zurück fahren *)
		IF fb_state_entry.E THEN
			zyl_rafo_vorschub.st_ctrl.in.b_einfahren := TRUE;
		END_IF

		(*-----------------------Weiterschaltbedingungen----------------------------*)
		IF zyl_rafo_vorschub.st_ctrl.out.b_eingefahren AND gb_ba_auto_kontroller THEN
			zyl_rafo_vorschub.st_ctrl.in.b_einfahren := FALSE;
			fb_state_entry.i16_next_step := 290;
		END_IF

(*=======================================================*)
	FEHLER:
		IF fb_state_entry.E THEN
			st_ctrl_out.b_fehler := TRUE;
			fb_ton_quitt.IN := FALSE;
			zyl_rafo_faenger.st_ctrl.in.b_quittieren := FALSE;
			zyl_rafo_klemmen.st_ctrl.in.b_quittieren := FALSE;
			zyl_rafo_vorschub.st_ctrl.in.b_quittieren := FALSE;
		END_IF

		(*-----------------------Weiterschaltbedingungen----------------------------*)
		IF st_ctrl_in.b_quitt AND NOT fb_state_entry.E THEN
			st_ctrl_out.b_fehler := FALSE;
			zyl_rafo_faenger.st_ctrl.in.b_quittieren := TRUE;
			zyl_rafo_klemmen.st_ctrl.in.b_quittieren := TRUE;
			zyl_rafo_vorschub.st_ctrl.in.b_quittieren := TRUE;
			fb_ton_quitt.IN := TRUE;
		END_IF

		IF fb_ton_quitt.Q THEN
			fb_ton_quitt.IN := FALSE;
			fb_state_entry.i16_next_step := INIT;
		END_IF

(*=======================================================*)
	STOP:
		IF fb_state_entry.E THEN
			fb_ton_quitt.IN := FALSE;
		END_IF

		(*-----------------------Weiterschaltbedingungen----------------------------*)
		IF st_ctrl_in.b_quitt AND NOT fb_state_entry.E THEN
			fb_ton_quitt.IN := TRUE;
		END_IF

		IF fb_ton_quitt.Q THEN
			fb_ton_quitt.IN := FALSE;
			fb_state_entry.i16_next_step := INIT;
		END_IF
END_CASE

fb_state_entry(
	i16_next_step:= , 
	i16_pos:= 2,
	s_debugtext:= ,
	E=> , 
	X=> , 
	i16_step=> ,
	i16_last_step=> );

IF st_config.b_config_fertig THEN
	(* Fehlermeldungen und Betriebsmeldungen ab dem Startindex in die globalen Meldungsarrays schreiben *)
	garr_stoermeldungen[st_config.i16_meld_startindex + 0] := sm_fehler_rafo_vorschub;
	garr_stoermeldungen[st_config.i16_meld_startindex + 1] := sm_keine_rafo_im_einzug;
	garr_stoermeldungen[st_config.i16_meld_startindex + 2] := FALSE;
	garr_stoermeldungen[st_config.i16_meld_startindex + 3] := FALSE;
	garr_stoermeldungen[st_config.i16_meld_startindex + 4] := FALSE;
	garr_stoermeldungen[st_config.i16_meld_startindex + 5] := FALSE;
	garr_stoermeldungen[st_config.i16_meld_startindex + 6] := FALSE;
	garr_stoermeldungen[st_config.i16_meld_startindex + 7] := FALSE;
	garr_stoermeldungen[st_config.i16_meld_startindex + 8] := FALSE;
	garr_stoermeldungen[st_config.i16_meld_startindex + 9] := FALSE;
	garr_stoermeldungen[st_config.i16_meld_startindex + 10] := FALSE;
	garr_stoermeldungen[st_config.i16_meld_startindex + 11] := FALSE;
	garr_stoermeldungen[st_config.i16_meld_startindex + 12] := FALSE;
	garr_stoermeldungen[st_config.i16_meld_startindex + 13] := FALSE;
	garr_stoermeldungen[st_config.i16_meld_startindex + 14] := FALSE;
	garr_stoermeldungen[st_config.i16_meld_startindex + 15] := FALSE;
	garr_stoermeldungen[st_config.i16_meld_startindex + 16] := FALSE;
	garr_stoermeldungen[st_config.i16_meld_startindex + 17] := FALSE;
	garr_stoermeldungen[st_config.i16_meld_startindex + 18] := FALSE;
	garr_stoermeldungen[st_config.i16_meld_startindex + 19] := FALSE;
	
	garr_betriebsmeldungen[st_config.i16_meld_startindex + 0] := FALSE;
	garr_betriebsmeldungen[st_config.i16_meld_startindex + 1] := FALSE;
	garr_betriebsmeldungen[st_config.i16_meld_startindex + 2] := FALSE;
	garr_betriebsmeldungen[st_config.i16_meld_startindex + 3] := FALSE;
	garr_betriebsmeldungen[st_config.i16_meld_startindex + 4] := FALSE;
	garr_betriebsmeldungen[st_config.i16_meld_startindex + 5] := FALSE;
	garr_betriebsmeldungen[st_config.i16_meld_startindex + 6] := FALSE;
	garr_betriebsmeldungen[st_config.i16_meld_startindex + 7] := FALSE;
	garr_betriebsmeldungen[st_config.i16_meld_startindex + 8] := FALSE;
	garr_betriebsmeldungen[st_config.i16_meld_startindex + 9] := FALSE;
	garr_betriebsmeldungen[st_config.i16_meld_startindex + 10] := FALSE;
	garr_betriebsmeldungen[st_config.i16_meld_startindex + 11] := FALSE;
	garr_betriebsmeldungen[st_config.i16_meld_startindex + 12] := FALSE;
	garr_betriebsmeldungen[st_config.i16_meld_startindex + 13] := FALSE;
	garr_betriebsmeldungen[st_config.i16_meld_startindex + 14] := FALSE;
	garr_betriebsmeldungen[st_config.i16_meld_startindex + 15] := FALSE;
	garr_betriebsmeldungen[st_config.i16_meld_startindex + 16] := FALSE;
	garr_betriebsmeldungen[st_config.i16_meld_startindex + 17] := FALSE;
	garr_betriebsmeldungen[st_config.i16_meld_startindex + 18] := FALSE;
	garr_betriebsmeldungen[st_config.i16_meld_startindex + 19] := FALSE;
END_IF
END_PROGRAM

(* POU Gemeinsamkeiten17xx/TagReader/ST_Konvertiere_gelese_TagData, ST *)
PROGRAM ST_Konvertiere_gelese_TagData
VAR
	i : INT := 0;
END_VAR
IF gst_datensatz.st_md.i16_tag_data_structur_version = 0 THEN
	gst_tag_data.WpcNumber := balluff_tag_reader.fb.s_lese_daten[0];
	gst_tag_data.StateParts[0] := balluff_tag_reader.fb.s_lese_daten[1];
	gst_tag_data.StateParts[1] := balluff_tag_reader.fb.s_lese_daten[2];

	MEMCPY( ADR(gst_tag_data.Articelnumber), ADR(balluff_tag_reader.fb.s_lese_daten[3]), 50);
	gst_tag_data.LastUsedTool := balluff_tag_reader.fb.s_lese_daten[54];
	MEMCPY( ADR(gst_tag_data.UmlNo_VPE), ADR(balluff_tag_reader.fb.s_lese_daten[55]), 4);
	gst_datensatz.st_md.s_aktuelle_artikelnummer := gst_tag_data.Articelnumber;
ELSIF gst_datensatz.st_md.i16_tag_data_structur_version = 1 THEN
	gst_tag_data.WpcNumber := balluff_tag_reader.fb.s_lese_daten[0];
	FOR i:= 0 TO 7 BY 1 DO
		gst_tag_data.StateParts[i] := balluff_tag_reader.fb.s_lese_daten[i + 1];
	END_FOR
	gst_tag_data.AmountPartsOnWpc := balluff_tag_reader.fb.s_lese_daten[10];
	gst_tag_data.LastUsedTool := balluff_tag_reader.fb.s_lese_daten[15];
	MEMCPY( ADR(gst_tag_data.Articelnumber), ADR(balluff_tag_reader.fb.s_lese_daten[20]), 50);
	MEMCPY( ADR(gst_tag_data.UmlNo_VPE), ADR(balluff_tag_reader.fb.s_lese_daten[71]), 4);
	gst_datensatz.st_md.s_aktuelle_artikelnummer := gst_tag_data.Articelnumber;
END_IF

(* Wenn Haken in Visu gesetzt ist dann BESTUECKUNG_MANUAL *)
(* Sonst kommt Info von der WT-XML *)
IF gst_datensatz.st_md.b_bestueckprogramm_manuell THEN
	gst_datensatz.st_md.i16_typ_bestueckmodus := BESTUECKUNG_MANUAL;
ELSE
	gst_datensatz.st_md.i16_typ_bestueckmodus := gst_datensatz.st_wt.i16_typ_bestueckmodus;
END_IF

(* Wenn Hublift links aktiv ist, soll Zelle Last Used Tool auf 0 zurücksetzen *)
(* Damit wird UML simuliert. Diese Funktion ermöglicht Kleinserien mit Hublift links *)
IF gst_datensatz.st_md.b_hublift_links_aktiv THEN
	gst_tag_data.StateParts[0] := PART_NEW;
	gst_tag_data.StateParts[1] := PART_NEW;
	gst_tag_data.LastUsedTool := 0;
END_IF
END_PROGRAM

(* POU Gemeinsamkeiten17xx/Achsen/ST_Virtuelle_Masterachse, ST *)
PROGRAM ST_Virtuelle_Masterachse
VAR_INPUT
	st_config_achse							: struct_ecd_config;
	e_ls_bandende_re				         		: BOOL;
	e_ls_bandende_li							: BOOL;
	st_ctrl_in									: struct_ctrl_in;
	e_steuerung_ein							: BOOL;
	e_ba_mit_bedingungen					: BOOL;
END_VAR
VAR_IN_OUT
	st_visu									: struct_ecd_visu;
	st_visu_virtuell							: struct_ecd_visu;
END_VAR
VAR_OUTPUT
	st_ctrl_out								: struct_ctrl_out;
	b_materialmangel							: BOOL;
	b_materialmangel2						: BOOL;
END_VAR
VAR
	st_sm						 			: struct_ecd_meldungen;
	st_drive_cmd								: struct_ecd_cmd;
	st_drive_cmd_bestueckachse				: struct_ecd_cmd;
	st_drive_cmd_z_achse						: struct_ecd_cmd;
	st_drive_cmd_y_achse						: struct_ecd_cmd;
	st_drive_cmd_b_achse						: struct_ecd_cmd;
	st_drive_cmd_virtuell						: struct_ecd_cmd;
	fb_ton_wz								: TON;
	fb_ton_quitt								: TON;
	fb_ton_wz_disable							: TON;
	fb_r_trig_tippen							: R_TRIG;
	fb_f_trig_tippen							: F_TRIG;
	fb_r_trig_start								: R_TRIG;
	fb_r_trig_start_remove_pos					: R_TRIG;
	fb_virt_master_axis						: ST_AxisJobCtrl_Motion;
	fb_axis_bestueckachse					: ST_AxisJobCtrl_Cam_Gear;
	fb_axis_z_achse							: ST_AxisJobCtrl_Cam_Gear;
	fb_axis_y_achse							: ST_AxisJobCtrl_Cam_Gear;
	fb_axis_b_achse							: ST_AxisJobCtrl_Cam_Gear;
	fb_state_entry								: ST_StateEntry;
	fb_ton_uez								: TON;
	fb_ton_pm_speed							: TON;
	fb_r_trig_pm_speed							: R_TRIG;
	i, j										: INT := 0;
	bm_an_visu_hinten						: STRING[255] := '';
	b_automatischer_bandwechsel				: BOOL := FALSE;
	b_bestueckschieber_ueberwachung_aktiv 	: BOOL := FALSE;
	b_einfaedeln_aktiv_servo					: BOOL := FALSE;	(* wenn TRUE dann entlüftet Serovbandeinzug nicht *)
	lr_merker_z_pos							: LREAL := 0.0;
	lr_merker_y_pos							: LREAL := 0.0;
	lr_merker_z_pos_alt						: LREAL := 0.0;
	lr_merker_z_pos_neu						: LREAL := 0.0;
	lr_merker_y_pos_alt						: LREAL := 0.0;
	lr_merker_y_pos_neu						: LREAL := 0.0;
	lr_abstand_yz								: LREAL := 0.0;
	lr_ErsteBestueckposY						: LREAL := 0.0;
	i16_merker_last_state						: INT := 0;
	i16_state_msg								:INT;
	fb_tof_bandende_li						: TOF;
	fb_tof_bandende_re						: TOF;
	fb_tof_bandende_rafo					: TOF;

	sm_fehler_bestueckanzahl					: BOOL := FALSE;
	sm_fehler_bestueckposition_z				: BOOL := FALSE;
	sm_fehler_bestueckposition_y				: BOOL := FALSE;
	sm_fehler_positionierung_z					: BOOL := FALSE;
	sm_fehler_positionierung_y					: BOOL := FALSE;
	sm_fehler_achse_lueften					: BOOL := FALSE;
	sm_fehler_raster_oder_zaehne				: BOOL := FALSE;
	sm_fehler_bestueckschieberanzahl			: BOOL := FALSE;
	sm_keine_busverbindung					: BOOL := FALSE;
	sm_fehler_nach_bandwechsel				: BOOL := FALSE;	(* Dieser Fehler soll kommen, damit Bediener Chargennummer des Bandes ins LTS einträgt, Wunsch von Sebastian Hechenrieder 27.11.17 *)
	sm_fehler_positionierung_bestueckachse		: BOOL := FALSE;

	(* Betriebsmeldungen *)
	bm_bandende_einzug_links_erreicht			: BOOL := FALSE;
	bm_bandende_einzug_rechts_erreicht		: BOOL := FALSE;
	bm_bandende_beide_einzuege_erreicht		: BOOL := FALSE;
	bm_einzug_links_band_entnehmen			: BOOL := FALSE;
	bm_einzug_links_band_auf_anschlag		: BOOL := FALSE;
	bm_einzug_rechts_band_entnehmen			: BOOL := FALSE;
	bm_einzug_rechts_band_auf_anschlag		: BOOL := FALSE;
	bm_override_kleiner_stufe9					: BOOL := FALSE;
	bm_einzug_rechts_band_bis_gls			: BOOL := FALSE;
	bm_einzug_links_band_bis_gls				: BOOL := FALSE;
	bm_beide_Bandklemmen_oeffnen			: BOOL := FALSE;
	bm_md_offset_z_pos_0_zu_hoch 			: BOOL := FALSE;
	bm_md_offset_y_pos_0_zu_hoch 			: BOOL := FALSE;

	b_merker_bandende_links					: BOOL := FALSE;
	b_merker_bandende_rechts				: BOOL := FALSE;
	b_hand_dialog_aktiv						: BOOL := FALSE;
	fb_r_trig_bestueckhubzaehler				: R_TRIG;
	fb_r_trig_skalierungsnocken					: R_TRIG;
	fb_f_trig_skalierungsnocken					: F_TRIG;
	fb_f_trig_ot								: F_TRIG;
	fb_r_trig_nockenumschaltung				: R_TRIG;
	err_id									: DWORD := 0;
	i16_bestueckachse_cam_table_id			: INT := 0;
	i16_bestueckachse_cam_table_id_alt		: INT := 0;

	fb_berechnung_override_achse				: ST_BerechnungOverride;

	i16_bestueckposzaehler					: INT := 0;

	i16_anzahl								: INT := 0;
	i16_einfaedelzaehler						: INT := 0;

	st_geschwindigkeiten						: struct_ecd_geschwindigkeiten;
	lr_decceleration_nothalt					: LREAL;
	lr_decceleration_normal					: LREAL;

	(* Lueften *)
	i16_step_lueften							: INT := 0;
	fb_r_trig_bandeinzug_lueften				: R_TRIG;
	fb_f_trig_bandeinzug_lueften				: F_TRIG;

	i16_LeftPins							: INT;
END_VAR
VAR CONSTANT
	r_auto_einfaedeln							: LREAL := 300.0;
	lr_faktor_override_reduzierung				: LREAL := 0.0025;
END_VAR
(* Zeiten *)
fb_ton_wz(IN:= ,PT:= , Q=>  , ET=> );
fb_ton_uez(IN:= ,	PT:= , Q=>  , ET=> );
fb_ton_quitt(IN:= , PT:= t#100ms, Q=> , ET=> );
fb_ton_wz_disable(IN:= , PT:= t#500ms, Q=> , ET=> );
fb_ton_pm_speed(IN:= , PT:= t#1h, Q=> , ET=> );

(* Flanken *)
fb_r_trig_skalierungsnocken(CLK:= nockenschaltwerk_bestueckachse.fb.arr_spur[SP_START_SKALIERUNG], Q=> );
fb_f_trig_skalierungsnocken(CLK:= nockenschaltwerk_bestueckachse.fb.arr_spur[SP_START_SKALIERUNG], Q=> );
fb_r_trig_start(CLK:= st_ctrl_in.b_start, Q=> );
fb_r_trig_bestueckhubzaehler(CLK:= nockenschaltwerk_bestueckachse.fb.arr_spur[SP_BESTUECKSCHIEBERHUB ], Q=> );
fb_f_trig_ot(CLK:= nockenschaltwerk_bestueckachse.fb.arr_spur[SP_OT], Q=> );
fb_r_trig_nockenumschaltung(CLK:= nockenschaltwerk_bestueckachse.fb.arr_spur[SP_BW_BESTUECKSCHIEBER_EINSTEUERN], Q=> );
fb_r_trig_start_remove_pos(CLK:= visu.b_start_remove_pos, Q=> );

(* Bandende Entprellen *)
fb_tof_bandende_li(IN:= e_ls_bandende_li , PT:=t#1100ms , Q=>  , ET=> );
fb_tof_bandende_re(IN:=e_ls_bandende_re , PT:=t#1100ms , Q=>  , ET=> );
fb_tof_bandende_rafo(IN:=ST_Rasterfolieneinzug.e_rasfo_ende , PT:=t#1100ms , Q=>  , ET=> );

(*Bei der Rasterfolie soll die Hubzahlreduzierung nicht angewendet werden*)
IF gst_datensatz.st_md.i16_typ_zelle <> RASTERFOLIE THEN
	fb_berechnung_override_achse.lr_FaktorHub := ST_BBGen.lr_FaktorHub;
ELSE
	fb_berechnung_override_achse.lr_FaktorHub := 1;
END_IF

(* Der Override der Virtuellen Masterachse wird an die zu fahrende Wegstrecke der Z-Achse angepasst *)
fb_berechnung_override_achse(
	lr_faktor := lr_faktor_override_reduzierung,
	i16_betriebsart:= gi16_betriebsart,
	lr_skalierung_slave_achse1:= ,
	lr_skalierung_slave_achse2:= ,
	lr_HubAuto:=gst_datensatz.st_wkz.r_auto,
	lr_override_vorgabe:= ST_TippTasten.lr_override_gestuft,
	lr_override=> );

(*Beim Einfädeln soll eine feste Geschwindigkeit verwendet werden*)
IF ST_TippTasten.b_einfaedeln_aktiv OR ST_TippTasten.b_initialisierungsphase THEN
	fb_virt_master_axis.lr_soll_geschwindigkeit := r_auto_einfaedeln;
ELSE
	fb_virt_master_axis.lr_soll_geschwindigkeit := gst_datensatz.st_wkz.r_auto;
END_IF

(* Achse steuern *)
(* Virtuelle Masterachse/Leitachse für die Bestückzelle*)
fb_virt_master_axis(
	e_referenznocken:= ,
	b_refsensor_vorhanden:= st_config_achse.b_refsensor_vorhanden,
	b_limitsensor_positiv_vorhanden:= st_config_achse.b_limitsensor_positiv_vorhanden,
	b_limitsensor_negativ_vorhanden:= st_config_achse.b_limitsensor_negativ_vorhanden,
	i16_achstyp := st_config_achse.i16_achstyp,
	lr_override_vorgabe := fb_berechnung_override_achse.lr_override,
	st_position:= ,
	mc_richtung_modulo:= ,
	mc_richtung_velocity:= ,
	mc_referenzmodus:= ,
	mc_buffermode_axis:= ,
	ui16_soeparam_write_value:= ,
	w_idn:= ,
	i16_nc_parameter_nummer:= ,
	r_wert_nc_write_parameter:= ,
	st_vorgabe_geschwindigkeiten:= st_geschwindigkeiten,
	b_bedingung_sls:= ,
	st_ads_info := ,
	st_eccoe_sdo := ,
	st_masterachse:= virtuelle_master_achse,
	st_visu_axis:= st_visu,
	st_ecd_cmd:= st_drive_cmd,
	ui16_soeparam_read_value=> ,
	r_wert_nc_read_parameter=> );

(* Entkoppeln der Slaveachsen bei Handbetrieb *)
IF gi16_betriebsart = HAND THEN
	(* Bei manuellem Fahren der Slaveachsen, muss diese erst entkoppelt werden *)
	IF ST_Bestueckachse.b_hand_dialog_aktiv AND bestueckachse.NcToPlc.CoupleState > 0 THEN
		st_drive_cmd_bestueckachse.enu_cmd := CAM_OUT_SLAVE;
	END_IF
	IF ST_Z_Achse.b_hand_dialog_aktiv AND z_achse.NcToPlc.CoupleState > 0 THEN
		st_drive_cmd_z_achse.enu_cmd := CAM_OUT_SLAVE;
	END_IF
	IF ST_Y_Achse.b_hand_dialog_aktiv AND y_achse.NcToPlc.CoupleState > 0 THEN
		st_drive_cmd_y_achse.enu_cmd := CAM_OUT_SLAVE;
	END_IF
	IF ST_Servobandeinzug.b_hand_dialog_aktiv AND b_achse.NcToPlc.CoupleState > 0 THEN
		st_drive_cmd_b_achse.enu_cmd := CAM_OUT_SLAVE;
	END_IF
END_IF

(* Bei betätigen der Bremse am hinteren Panel muss die Master-Slave-Kopplung gelöst werden. *)
IF visu_hinten.out.ST_Servobandeinzug.b_taste_bremse AND b_achse.NcToPlc.CoupleState > 0 THEN
	st_drive_cmd_b_achse.enu_cmd := CAM_OUT_SLAVE;
END_IF

(* Override kleiner als Stufe 10 dann Meldelampe*)
IF	ST_TippTasten.i16_akt_stufe<>9 AND gst_datensatz.st_md.i16_typ_bestueckmodus<>BESTUECKUNG_MANUAL THEN
	b_materialmangel :=TRUE;
	bm_override_kleiner_stufe9:= TRUE;
	fb_ton_pm_speed.IN := TRUE;
ELSE
	b_materialmangel :=FALSE;
	bm_override_kleiner_stufe9:= FALSE;
	fb_ton_pm_speed.IN := FALSE;
END_IF

fb_r_trig_pm_speed(CLK:= fb_ton_pm_speed.Q, Q=> );

IF fb_r_trig_pm_speed.Q THEN
	i16_state_msg := 1;
END_IF

(*Produktionsmeldung für Geschwindigkeit zu niedrig*)
CASE i16_state_msg OF
	1: (*Warten bis keine ander Produktions Meldung ansteht *)
		IF	TestAndSet(ST_Message_Produktion.LockFlag) THEN
			ST_Message_Produktion.ClearMessageLines();
			i16_state_msg := 2;
		END_IF

	2:  (*Produktions Meldung*)
		Visu.MeldungProduktion.Color_R := 255;
		Visu.MeldungProduktion.Color_G := 255;
		Visu.MeldungProduktion.Color_B := 0;
		IF visu.s_akt_sprache = 'de' THEN
			Visu.MeldungProduktion.Name:='Geschwindigkeit zu niedrig eingestellt.';
		ELSIF visu.s_akt_sprache = 'en' THEN
			Visu.MeldungProduktion.Name:='stiching speed is set too low.';
		ELSIF visu.s_akt_sprache = 'cz' THEN
			Visu.MeldungProduktion.Name:='Rychlost osazovani je priliz nizka.';
		END_IF
		Visu.MeldungProduktion.ShowMessage := TRUE;
		Visu.MeldungProduktion.Button1.sichtbar:=TRUE;	(*OK*)
		Visu.MeldungProduktion.Button1.Text:='Ok';
		i16_state_msg := 3;

	3:  (*Warte auf OK*)
		IF Visu.MeldungProduktion.Button1.tasten THEN
			i16_state_msg:=0;
			fb_ton_pm_speed.IN := FALSE;
		END_IF
END_CASE

(* Korrekturwerte für X- und Z- Achse sind zu hoch *)
IF ABS(gst_datensatz.st_md.lr_offset_z_pos_0) > 0.5 THEN
	bm_md_offset_z_pos_0_zu_hoch := TRUE;
ELSE
	bm_md_offset_z_pos_0_zu_hoch := FALSE;
END_IF

IF ABS(gst_datensatz.st_md.lr_offset_y_pos_0) > 0.5 THEN
	bm_md_offset_y_pos_0_zu_hoch := TRUE;
ELSE
	bm_md_offset_y_pos_0_zu_hoch := FALSE;
END_IF

IF bm_md_offset_z_pos_0_zu_hoch OR bm_md_offset_y_pos_0_zu_hoch THEN
	b_materialmangel2 := TRUE;
ELSE
	b_materialmangel2 := FALSE;
END_IF

(* Hinweis: Die Y-Achse darf nur dann in den Slavebetrieb mit der Bestückachse gehen, wenn diese nicht als Slave an die Z-Achse gekoppelt ist. *)
(* Ansonsten kommt es zum Fehler, weil eine Slaveachse nicht gleichzeitig an zwei Masterachsen gekoppelt werden kann!  *)
CASE gst_datensatz.st_md.i16_typ_zelle OF
	KEINE_ZELLE:
		;

	BESTUECKZELLE_1700,  RASTERFOLIE:
		IF bestueckachse.NcToPlc.CoupleState > 0 OR st_drive_cmd_bestueckachse.enu_cmd > NO_COMMAND THEN
			(* Slave Bestückachse *)
			fb_axis_bestueckachse.st_camin_options.CamOperationMode := CAMOPERATIONMODE_EXCHANGE;
			fb_axis_bestueckachse.st_camscaling_data.MasterScalingMode := MC_CAMSCALING_OFF;
			fb_axis_bestueckachse.st_camscaling_data.SlaveScalingMode := MC_CAMSCALING_AUTOOFFSET;
			(* Kurvenscheibenkopplung ein/ausschalten *)
			fb_axis_bestueckachse(
				r_getriebefaktor := 1.0,
				r_master_position:= ,
				mc_activation_mode_camin:= ,
				lr_activation_position_camin:= ,
				mc_activation_mode_scaleing:= ,
				lr_activation_position_scaleing:= ,
				mc_buffermode_axis:= ,
				mc_cam_table_id:=  i16_bestueckachse_cam_table_id,
				mc_cam_point_id:= ,
				mc_motion_function_point:= ,
				st_camin_options:= ,
				st_camexchange_options:= ,
				mc_reference_cam_table_id:= ,
				st_camscaling_data:= ,
				st_masterachse:= virtuelle_master_achse,
				st_slaveachse:= bestueckachse,
				st_ecd_cmd:= st_drive_cmd_bestueckachse);
		END_IF

		IF z_achse.NcToPlc.CoupleState > 0 OR st_drive_cmd_z_achse.enu_cmd > NO_COMMAND THEN
			(* Slave Z-Achse *)
			fb_axis_z_achse.st_camscaling_data.SlaveRelative := TRUE;
			(* Kurvenscheibenkopplung ein/ausschalten *)
			fb_axis_z_achse(
				r_getriebefaktor:= 1.0,
				r_master_position:= ,
				mc_activation_mode_camin:= MC_CAMACTIVATION_INSTANTANEOUS,
				lr_activation_position_camin:= 0.0,
				mc_activation_mode_scaleing:= MC_CAMACTIVATION_INSTANTANEOUS,
				lr_activation_position_scaleing:= 0.0,
				mc_buffermode_axis:= ,
				mc_cam_table_id:=  1,
				mc_cam_point_id:= ,
				mc_motion_function_point:= ,
				st_camin_options:= ,
				st_camexchange_options:= ,
				mc_reference_cam_table_id:= ,
				st_camscaling_data:= ,
				st_masterachse:= virtuelle_master_achse,
				st_slaveachse:= z_achse,
				st_ecd_cmd:= st_drive_cmd_z_achse );
		END_IF

		(* Fallunterscheidung Bandeinzug *)
		CASE gst_datensatz.st_wkz.i16_typ_bandeinzug OF
			KEIN_EINZUG:
				;
			STANDARD_2FACH_V2:
				;
			BANDWECHSLER_V2:
				;
			SERVO:
				(* Slave B-Achse *)
				fb_axis_b_achse.st_camscaling_data.SlaveRelative := TRUE;
				(* Kurvenscheibenkopplung ein/ausschalten *)
				fb_axis_b_achse(
					r_getriebefaktor:= 1.0,
					r_master_position:= ,
					mc_activation_mode_camin:= MC_CAMACTIVATION_INSTANTANEOUS,
					lr_activation_position_camin:= 0.0,
					mc_activation_mode_scaleing:= MC_CAMACTIVATION_INSTANTANEOUS,
					lr_activation_position_scaleing:= 0.0,
					mc_buffermode_axis:= ,
					mc_cam_table_id:=  4,
					mc_cam_point_id:= ,
					mc_motion_function_point:= ,
					st_camin_options:= ,
					st_camexchange_options:= ,
					mc_reference_cam_table_id:= ,
					st_camscaling_data:= ,
					st_masterachse:= bestueckachse,
					st_slaveachse:= b_achse,
					st_ecd_cmd:= st_drive_cmd_b_achse );
		END_CASE

		IF y_achse.NcToPlc.CoupleState > 0 OR st_drive_cmd_y_achse.enu_cmd > NO_COMMAND THEN
			(* Slave Y-Achse *)
			fb_axis_y_achse.st_camscaling_data.SlaveRelative := TRUE;
			(* Kurvenscheibenkopplung ein/ausschalten *)
			fb_axis_y_achse(
				r_getriebefaktor:= 1.0,
				r_master_position:= ,
				mc_activation_mode_camin:= MC_CAMACTIVATION_INSTANTANEOUS,
				lr_activation_position_camin:= 0.0,
				mc_activation_mode_scaleing:= MC_CAMACTIVATION_INSTANTANEOUS,
				lr_activation_position_scaleing:= 0.0,
				mc_buffermode_axis:= ,
				mc_cam_table_id:= 3 ,
				mc_cam_point_id:= ,
				mc_motion_function_point:= ,
				st_camin_options:= ,
				st_camexchange_options:= ,
				mc_reference_cam_table_id:= ,
				st_camscaling_data:= ,
				st_masterachse:= virtuelle_master_achse,
				st_slaveachse:= y_achse,
				st_ecd_cmd:= st_drive_cmd_y_achse );
		END_IF

	BESTUECKZELLE_1720:
		IF bestueckachse.NcToPlc.CoupleState > 0 OR st_drive_cmd_bestueckachse.enu_cmd > NO_COMMAND THEN
			(* Slave Bestückachse *)
			fb_axis_bestueckachse.st_camin_options.CamOperationMode := CAMOPERATIONMODE_EXCHANGE;
			fb_axis_bestueckachse.st_camscaling_data.MasterScalingMode := MC_CAMSCALING_OFF;
			fb_axis_bestueckachse.st_camscaling_data.SlaveScalingMode := MC_CAMSCALING_OFF;
			(* Kurvenscheibenkopplung ein/ausschalten *)
			fb_axis_bestueckachse(
				r_getriebefaktor := 1.0,
				r_master_position:= ,
				mc_activation_mode_camin:= ,
				lr_activation_position_camin:= ,
				mc_activation_mode_scaleing:= ,
				lr_activation_position_scaleing:= ,
				mc_buffermode_axis:= ,
				mc_cam_table_id:=  i16_bestueckachse_cam_table_id,
				mc_cam_point_id:= ,
				mc_motion_function_point:= ,
				st_camin_options:= ,
				st_camexchange_options:= ,
				mc_reference_cam_table_id:= ,
				st_camscaling_data:= ,
				st_masterachse:= virtuelle_master_achse,
				st_slaveachse:= bestueckachse,
				st_ecd_cmd:= st_drive_cmd_bestueckachse);
		END_IF

		IF z_achse.NcToPlc.CoupleState > 0 OR st_drive_cmd_z_achse.enu_cmd > NO_COMMAND THEN
			(* Slave Z-Achse *)
			fb_axis_z_achse.st_camscaling_data.SlaveRelative := TRUE;
			(* Kurvenscheibenkopplung ein/ausschalten *)
			fb_axis_z_achse(
				r_getriebefaktor:= 1.0,
				r_master_position:= ,
				mc_activation_mode_camin:= MC_CAMACTIVATION_INSTANTANEOUS,
				lr_activation_position_camin:= 0.0,
				mc_activation_mode_scaleing:= MC_CAMACTIVATION_INSTANTANEOUS,
				lr_activation_position_scaleing:= 0.0,
				mc_buffermode_axis:= ,
				mc_cam_table_id:=  1,
				mc_cam_point_id:= ,
				mc_motion_function_point:= ,
				st_camin_options:= ,
				st_camexchange_options:= ,
				mc_reference_cam_table_id:= ,
				st_camscaling_data:= ,
				st_masterachse:= virtuelle_master_achse,
				st_slaveachse:= z_achse,
				st_ecd_cmd:= st_drive_cmd_z_achse );
		END_IF

END_CASE

(* Bandeinzug lüften-regeln *)
subr_ST_EinzugLueften();

(* =======================================Toplevel========================================== *)
(* =====Achse wird disabled===== *)
IF (NOT e_steuerung_ein OR NOT e_ba_mit_bedingungen) AND bestueckachse.Status.Operational THEN
	st_drive_cmd.enu_cmd := POWER_DISABLE;
END_IF

IF fb_state_entry.i16_next_step > INIT AND fb_state_entry.i16_next_step < FEHLER THEN
	(* =====Fehler vom Achskontroller===== *)
	IF	st_drive_cmd.b_job_fehler OR
		st_drive_cmd_bestueckachse.b_job_fehler OR
		st_drive_cmd_z_achse.b_job_fehler OR
		st_drive_cmd_y_achse.b_job_fehler OR
		st_drive_cmd_b_achse.b_job_fehler
		THEN
			fb_state_entry.i16_next_step := FEHLER;
	END_IF

	IF fb_state_entry.i16_next_step > 45 THEN
		(* Devicefehler *)
		IF virtuelle_master_achse.Status.Error THEN
			st_sm.b_achsfehler := TRUE;
			fb_state_entry.i16_next_step := FEHLER;
		ELSIF virtuelle_master_achse.Status.DriveDeviceError THEN
			st_sm.b_devicefehler := TRUE;
			fb_state_entry.i16_next_step := FEHLER;
		END_IF
	END_IF

	IF fb_state_entry.i16_next_step < STOP THEN
		(* =====Achse wird gestoppt===== *)
		IF st_ctrl_in.b_stop THEN
			fb_state_entry.i16_next_step := STOP;
		ELSIF fb_state_entry.i16_next_step < HALT THEN
			(* =====Achse wird angehalten===== *)
			IF st_ctrl_in.b_halt THEN
				fb_state_entry.i16_next_step := HALT;
			END_IF
		END_IF
	END_IF

END_IF

